DATA_BLOCK "FixReadCap_copy"
{ S7_Optimized_Access := 'FALSE' }
VERSION : 0.1
   STRUCT
      W0 : Int;   // M501_Z0 Destination_1A
      W2 : Int;   // M501_Z0 Destination_1B
      W4 : Int;   // M501_Z0 Destination_1C
      W6 : Int;   // M501_Z0 Destination_1D
      W8 : Int;   // M501_Z0 Length_1A (x) [dm]
      W10 : Int;   // M501_Z0 Length_1B (x) [dm]
      W12 : Int;   // M501_Z0 Length_1C (x) [dm]
      W14 : Int;   // M501_Z0 Length_1D (x) [dm]
      W16 : Int;   // M501_Z0 Width_1A  (y) [dm]
      W18 : Int;   // M501_Z0 Width_1B  (y) [dm]
      W20 : Int;   // M501_Z0 Width_1C  (y) [dm]
      W22 : Int;   // M501_Z0 Width_1D  (y) [dm]
      W24 : Int;   // M501_Z0 Position_X_1A  [dm]
      W26 : Int;   // M501_Z0 Position_X_1B  [dm]
      W28 : Int;   // M501_Z0 Position_X_1C  [dm]
      W30 : Int;   // M501_Z0 Position_X_1D  [dm]
      W32 : Int;   // M501_Z0 Position_Y_1A  [dm]
      W34 : Int;   // M501_Z0 Position_Y_1B  [dm]
      W36 : Int;   // M501_Z0 Position_Y_1C  [dm]
      W38 : Int;   // M501_Z0 Position_Y_1D  [dm]
      W40 : Int;   // M501_Z0 Code_1A_not used
      W42 : Int;   // M501_Z0 Code_1B_not used
      W44 : Int;   // M501_Z0 Code_1C_not used
      W46 : Int;   // M501_Z0 Code_1D_not used
      W48 : Int;
      W50 : Int;   // M501_Z1 Destination_1A
      W52 : Int;   // M501_Z1 Destination_1B
      W54 : Int;   // M501_Z1 Destination_1C
      W56 : Int;   // M501_Z1 Destination_1D
      W58 : Int;   // M501_Z1 Length_1A (x) [dm]
      W60 : Int;   // M501_Z1 Length_1B (x) [dm]
      W62 : Int;   // M501_Z1 Length_1C (x) [dm]
      W64 : Int;   // M501_Z1 Length_1D (x) [dm]
      W66 : Int;   // M501_Z1 Width_1A  (y) [dm]
      W68 : Int;   // M501_Z1 Width_1B  (y) [dm]
      W70 : Int;   // M501_Z1 Width_1C  (y) [dm]
      W72 : Int;   // M501_Z1 Width_1D  (y) [dm]
      W74 : Int;   // M501_Z1 Position_X_1A  [dm]
      W76 : Int;   // M501_Z1 Position_X_1B  [dm]
      W78 : Int;   // M501_Z1 Position_X_1C  [dm]
      W80 : Int;   // M501_Z1 Position_X_1D  [dm]
      W82 : Int;   // M501_Z1 Position_Y_1A  [dm]
      W84 : Int;   // M501_Z1 Position_Y_1B  [dm]
      W86 : Int;   // M501_Z1 Position_Y_1C  [dm]
      W88 : Int;   // M501_Z1 Position_Y_1D  [dm]
      W90 : Int;   // M501_Z1 Code_1A_not used
      W92 : Int;   // M501_Z1 Code_1B_not used
      W94 : Int;   // M501_Z1 Code_1C_not used
      W96 : Int;   // M501_Z1 Code_1D_not used
      W98 : Int;
      W100 : Int;   // M501_Z2 Destination_1A
      W102 : Int;   // M501_Z2 Destination_1B
      W104 : Int;   // M501_Z2 Destination_1C
      W106 : Int;   // M501_Z2 Destination_1D
      W108 : Int;   // M501_Z2 Length_1A (x) [dm]
      W110 : Int;   // M501_Z2 Length_1B (x) [dm]
      W112 : Int;   // M501_Z2 Length_1C (x) [dm]
      W114 : Int;   // M501_Z2 Length_1D (x) [dm]
      W116 : Int;   // M501_Z2 Width_1A  (y) [dm]
      W118 : Int;   // M501_Z2 Width_1B  (y) [dm]
      W120 : Int;   // M501_Z2 Width_1C  (y) [dm]
      W122 : Int;   // M501_Z2 Width_1D  (y) [dm]
      W124 : Int;   // M501_Z2 Position_X_1A  [dm]
      W126 : Int;   // M501_Z2 Position_X_1B  [dm]
      W128 : Int;   // M501_Z2 Position_X_1C  [dm]
      W130 : Int;   // M501_Z2 Position_X_1D  [dm]
      W132 : Int;   // M501_Z2 Position_Y_1A  [dm]
      W134 : Int;   // M501_Z2 Position_Y_1B  [dm]
      W136 : Int;   // M501_Z2 Position_Y_1C  [dm]
      W138 : Int;   // M501_Z2 Position_Y_1D  [dm]
      W140 : Int;   // M501_Z2 Code_1A_not used
      W142 : Int;   // M501_Z2 Code_1B_not used
      W144 : Int;   // M501_Z2 Code_1C_not used
      W146 : Int;   // M501_Z2 Code_1D_not used
      W148 : Int;
      W150 : Int;   // M319 Destination_1A
      W152 : Int;   // M319 Destination_2A
      W154 : Int;   // M319 Destination_3A
      W156 : Int;   // M319 Destination_4A
      W158 : Int;   // M319 Length_1A (x) [dm]
      W160 : Int;   // M319 Length_2A (x) [dm]
      W162 : Int;   // M319 Length_3A (x) [dm]
      W164 : Int;   // M319 Length_4A (x) [dm]
      W166 : Int;   // M319 Width_1A  (y) [dm]
      W168 : Int;   // M319 Width_2A  (y) [dm]
      W170 : Int;   // M319 Width_3A  (y) [dm]
      W172 : Int;   // M319 Width_4A  (y) [dm]
      W174 : Int;   // M319 Position_X_1A  [dm]
      W176 : Int;   // M319 Position_X_2A  [dm]
      W178 : Int;   // M319 Position_X_3A  [dm]
      W180 : Int;   // M319 Position_X_4A  [dm]
      W182 : Int;   // M319 Position_Y_1A  [dm]
      W184 : Int;   // M319 Position_Y_2A  [dm]
      W186 : Int;   // M319 Position_Y_3A  [dm]
      W188 : Int;   // M319 Position_Y_4A  [dm]
      W190 : Int;   // M319 Code_1A_not used
      W192 : Int;   // M319 Code_2A_not used
      W194 : Int;   // M319 Code_3A_not used
      W196 : Int;   // M319 Code_4A_not used
      W198 : Int;
      W200 : Int;   // M502 Destination_1A
      W202 : Int;   // M502 Destination_2A
      W204 : Int;   // M502 Destination_3A
      W206 : Int;   // M502 Destination_4A
      W208 : Int;   // M502 Length_1A (x) [dm]
      W210 : Int;   // M502 Length_2A (x) [dm]
      W212 : Int;   // M502 Length_3A (x) [dm]
      W214 : Int;   // M502 Length_4A (x) [dm]
      W216 : Int;   // M502 Width_1A  (y) [dm]
      W218 : Int;   // M502 Width_2A  (y) [dm]
      W220 : Int;   // M502 Width_3A  (y) [dm]
      W222 : Int;   // M502 Width_4A  (y) [dm]
      W224 : Int;   // M502 Position_X_1A  [dm]
      W226 : Int;   // M502 Position_X_2A  [dm]
      W228 : Int;   // M502 Position_X_3A  [dm]
      W230 : Int;   // M502 Position_X_4A  [dm]
      W232 : Int;   // M502 Position_Y_1A  [dm]
      W234 : Int;   // M502 Position_Y_2A  [dm]
      W236 : Int;   // M502 Position_Y_3A  [dm]
      W238 : Int;   // M502 Position_Y_4A  [dm]
      W240 : Int;   // M502 Code_1A_not used
      W242 : Int;   // M502 Code_2A_not used
      W244 : Int;   // M502 Code_3A_not used
      W246 : Int;   // M502 Code_4A_not used
      W248 : Int;
      W250 : Int;   // M502 Destination_1B
      W252 : Int;   // M502 Destination_2B
      W254 : Int;   // M502 Destination_3B
      W256 : Int;   // M502 Destination_4B
      W258 : Int;   // M502 Length_1B (x) [dm]
      W260 : Int;   // M502 Length_2B (x) [dm]
      W262 : Int;   // M502 Length_3B (x) [dm]
      W264 : Int;   // M502 Length_4B (x) [dm]
      W266 : Int;   // M502 Width_1B  (y) [dm]
      W268 : Int;   // M502 Width_2B  (y) [dm]
      W270 : Int;   // M502 Width_3B  (y) [dm]
      W272 : Int;   // M502 Width_4B  (y) [dm]
      W274 : Int;   // M502 Position_X_1B  [dm]
      W276 : Int;   // M502 Position_X_2B  [dm]
      W278 : Int;   // M502 Position_X_3B  [dm]
      W280 : Int;   // M502 Position_X_4B  [dm]
      W282 : Int;   // M502 Position_Y_1B  [dm]
      W284 : Int;   // M502 Position_Y_2B  [dm]
      W286 : Int;   // M502 Position_Y_3B  [dm]
      W288 : Int;   // M502 Position_Y_4B  [dm]
      W290 : Int;   // M502 Code_1B_not used
      W292 : Int;   // M502 Code_2B_not used
      W294 : Int;   // M502 Code_3B_not used
      W296 : Int;   // M502 Code_4B_not used
      W298 : Int;
      W300 : Int;   // M504 Destination_1A
      W302 : Int;   // M504 Destination_2A
      W304 : Int;   // M504 Destination_3A
      W306 : Int;   // M504 Destination_4A
      W308 : Int;   // M504 Length_1A (x) [dm]
      W310 : Int;   // M504 Length_2A (x) [dm]
      W312 : Int;   // M504 Length_3A (x) [dm]
      W314 : Int;   // M504 Length_4A (x) [dm]
      W316 : Int;   // M504 Width_1A  (y) [dm]
      W318 : Int;   // M504 Width_2A  (y) [dm]
      W320 : Int;   // M504 Width_3A  (y) [dm]
      W322 : Int;   // M504 Width_4A  (y) [dm]
      W324 : Int;   // M504 Position_X_1A  [dm]
      W326 : Int;   // M504 Position_X_2A  [dm]
      W328 : Int;   // M504 Position_X_3A  [dm]
      W330 : Int;   // M504 Position_X_4A  [dm]
      W332 : Int;   // M504 Position_Y_1A  [dm]
      W334 : Int;   // M504 Position_Y_2A  [dm]
      W336 : Int;   // M504 Position_Y_3A  [dm]
      W338 : Int;   // M504 Position_Y_4A  [dm]
      W340 : Int;   // M504 Code_1A_not used
      W342 : Int;   // M504 Code_2A_not used
      W344 : Int;   // M504 Code_3A_not used
      W346 : Int;   // M504 Code_4A_not used
      W348 : Int;
      W350 : Int;   // M504 Destination_1B
      W352 : Int;   // M504 Destination_2B
      W354 : Int;   // M504 Destination_3B
      W356 : Int;   // M504 Destination_4B
      W358 : Int;   // M504 Length_1B (x) [dm]
      W360 : Int;   // M504 Length_2B (x) [dm]
      W362 : Int;   // M504 Length_3B (x) [dm]
      W364 : Int;   // M504 Length_4B (x) [dm]
      W366 : Int;   // M504 Width_1B  (y) [dm]
      W368 : Int;   // M504 Width_2B  (y) [dm]
      W370 : Int;   // M504 Width_3B  (y) [dm]
      W372 : Int;   // M504 Width_4B  (y) [dm]
      W374 : Int;   // M504 Position_X_1B  [dm]
      W376 : Int;   // M504 Position_X_2B  [dm]
      W378 : Int;   // M504 Position_X_3B  [dm]
      W380 : Int;   // M504 Position_X_4B  [dm]
      W382 : Int;   // M504 Position_Y_1B  [dm]
      W384 : Int;   // M504 Position_Y_2B  [dm]
      W386 : Int;   // M504 Position_Y_3B  [dm]
      W388 : Int;   // M504 Position_Y_4B  [dm]
      W390 : Int;   // M504 Code_1B_not used
      W392 : Int;   // M504 Code_2B_not used
      W394 : Int;   // M504 Code_3B_not used
      W396 : Int;   // M504 Code_4B_not used
      W398 : Int;
      W400 : Int;   // M505 Destination_1A
      W402 : Int;   // M505 Destination_2A
      W404 : Int;   // M505 Destination_3A
      W406 : Int;   // M505 Destination_4A
      W408 : Int;   // M505 Length_1A (x) [dm]
      W410 : Int;   // M505 Length_2A (x) [dm]
      W412 : Int;   // M505 Length_3A (x) [dm]
      W414 : Int;   // M505 Length_4A (x) [dm]
      W416 : Int;   // M505 Width_1A  (y) [dm]
      W418 : Int;   // M505 Width_2A  (y) [dm]
      W420 : Int;   // M505 Width_3A  (y) [dm]
      W422 : Int;   // M505 Width_4A  (y) [dm]
      W424 : Int;   // M505 Position_X_1A  [dm]
      W426 : Int;   // M505 Position_X_2A  [dm]
      W428 : Int;   // M505 Position_X_3A  [dm]
      W430 : Int;   // M505 Position_X_4A  [dm]
      W432 : Int;   // M505 Position_Y_1A  [dm]
      W434 : Int;   // M505 Position_Y_2A  [dm]
      W436 : Int;   // M505 Position_Y_3A  [dm]
      W438 : Int;   // M505 Position_Y_4A  [dm]
      W440 : Int;   // M505 Code_1A_not used
      W442 : Int;   // M505 Code_2A_not used
      W444 : Int;   // M505 Code_3A_not used
      W446 : Int;   // M505 Code_4A_not used
      W448 : Int;
      W450 : Int;   // M505 Destination_1B
      W452 : Int;   // M505 Destination_2B
      W454 : Int;   // M505 Destination_3B
      W456 : Int;   // M505 Destination_4B
      W458 : Int;   // M505 Length_1B (x) [dm]
      W460 : Int;   // M505 Length_2B (x) [dm]
      W462 : Int;   // M505 Length_3B (x) [dm]
      W464 : Int;   // M505 Length_4B (x) [dm]
      W466 : Int;   // M505 Width_1B  (y) [dm]
      W468 : Int;   // M505 Width_2B  (y) [dm]
      W470 : Int;   // M505 Width_3B  (y) [dm]
      W472 : Int;   // M505 Width_4B  (y) [dm]
      W474 : Int;   // M505 Position_X_1B  [dm]
      W476 : Int;   // M505 Position_X_2B  [dm]
      W478 : Int;   // M505 Position_X_3B  [dm]
      W480 : Int;   // M505 Position_X_4B  [dm]
      W482 : Int;   // M505 Position_Y_1B  [dm]
      W484 : Int;   // M505 Position_Y_2B  [dm]
      W486 : Int;   // M505 Position_Y_3B  [dm]
      W488 : Int;   // M505 Position_Y_4B  [dm]
      W490 : Int;   // M505 Code_1B_not used
      W492 : Int;   // M505 Code_2B_not used
      W494 : Int;   // M505 Code_3B_not used
      W496 : Int;   // M505 Code_4B_not used
      W498 : Int;
      W500 : Int;   // M506 Destination_1A
      W502 : Int;   // M506 Destination_2A
      W504 : Int;   // M506 Destination_3A
      W506 : Int;   // M506 Destination_4A
      W508 : Int;   // M506 Length_1A (x) [dm]
      W510 : Int;   // M506 Length_2A (x) [dm]
      W512 : Int;   // M506 Length_3A (x) [dm]
      W514 : Int;   // M506 Length_4A (x) [dm]
      W516 : Int;   // M506 Width_1A  (y) [dm]
      W518 : Int;   // M506 Width_2A  (y) [dm]
      W520 : Int;   // M506 Width_3A  (y) [dm]
      W522 : Int;   // M506 Width_4A  (y) [dm]
      W524 : Int;   // M506 Position_X_1A  [dm]
      W526 : Int;   // M506 Position_X_2A  [dm]
      W528 : Int;   // M506 Position_X_3A  [dm]
      W530 : Int;   // M506 Position_X_4A  [dm]
      W532 : Int;   // M506 Position_Y_1A  [dm]
      W534 : Int;   // M506 Position_Y_2A  [dm]
      W536 : Int;   // M506 Position_Y_3A  [dm]
      W538 : Int;   // M506 Position_Y_4A  [dm]
      W540 : Int;   // M506 Code_1A_not used
      W542 : Int;   // M506 Code_2A_not used
      W544 : Int;   // M506 Code_3A_not used
      W546 : Int;   // M506 Code_4A_not used
      W548 : Int;
      W550 : Int;   // M506 Destination_1B
      W552 : Int;   // M506 Destination_2B
      W554 : Int;   // M506 Destination_3B
      W556 : Int;   // M506 Destination_4B
      W558 : Int;   // M506 Length_1B (x) [dm]
      W560 : Int;   // M506 Length_2B (x) [dm]
      W562 : Int;   // M506 Length_3B (x) [dm]
      W564 : Int;   // M506 Length_4B (x) [dm]
      W566 : Int;   // M506 Width_1B  (y) [dm]
      W568 : Int;   // M506 Width_2B  (y) [dm]
      W570 : Int;   // M506 Width_3B  (y) [dm]
      W572 : Int;   // M506 Width_4B  (y) [dm]
      W574 : Int;   // M506 Position_X_1B  [dm]
      W576 : Int;   // M506 Position_X_2B  [dm]
      W578 : Int;   // M506 Position_X_3B  [dm]
      W580 : Int;   // M506 Position_X_4B  [dm]
      W582 : Int;   // M506 Position_Y_1B  [dm]
      W584 : Int;   // M506 Position_Y_2B  [dm]
      W586 : Int;   // M506 Position_Y_3B  [dm]
      W588 : Int;   // M506 Position_Y_4B  [dm]
      W590 : Int;   // M506 Code_1B_not used
      W592 : Int;   // M506 Code_2B_not used
      W594 : Int;   // M506 Code_3B_not used
      W596 : Int;   // M506 Code_4B_not used
      W598 : Int;
      W600 : Int;
   END_STRUCT;


BEGIN
   W150 := 30;
   W158 := 36;
   W166 := 15;
   W168 := 15;
   W170 := 15;
   W172 := 15;
   W174 := 3;
   W176 := -34;
   W178 := -71;
   W180 := -108;
   W182 := 15;
   W184 := 15;
   W186 := 15;
   W188 := 15;
   W190 := 7255;
   W200 := 1;
   W206 := 30541;

END_DATA_BLOCK

DATA_BLOCK "FixReadCap"
{ S7_Optimized_Access := 'FALSE' }
VERSION : 0.1
   STRUCT
      W0 : Int;   // M501_Z0 Destination_1A
      W2 : Int;   // M501_Z0 Destination_1B
      W4 : Int;   // M501_Z0 Destination_1C
      W6 : Int;   // M501_Z0 Destination_1D
      W8 : Int;   // M501_Z0 Length_1A (x) [dm]
      W10 : Int;   // M501_Z0 Length_1B (x) [dm]
      W12 : Int;   // M501_Z0 Length_1C (x) [dm]
      W14 : Int;   // M501_Z0 Length_1D (x) [dm]
      W16 : Int;   // M501_Z0 Width_1A  (y) [dm]
      W18 : Int;   // M501_Z0 Width_1B  (y) [dm]
      W20 : Int;   // M501_Z0 Width_1C  (y) [dm]
      W22 : Int;   // M501_Z0 Width_1D  (y) [dm]
      W24 : Int;   // M501_Z0 Position_X_1A  [dm]
      W26 : Int;   // M501_Z0 Position_X_1B  [dm]
      W28 : Int;   // M501_Z0 Position_X_1C  [dm]
      W30 : Int;   // M501_Z0 Position_X_1D  [dm]
      W32 : Int;   // M501_Z0 Position_Y_1A  [dm]
      W34 : Int;   // M501_Z0 Position_Y_1B  [dm]
      W36 : Int;   // M501_Z0 Position_Y_1C  [dm]
      W38 : Int;   // M501_Z0 Position_Y_1D  [dm]
      W40 : Int;   // M501_Z0 Code_1A_not used
      W42 : Int;   // M501_Z0 Code_1B_not used
      W44 : Int;   // M501_Z0 Code_1C_not used
      W46 : Int;   // M501_Z0 Code_1D_not used
      W48 : Int;
      W50 : Int;   // M501_Z1 Destination_1A
      W52 : Int;   // M501_Z1 Destination_1B
      W54 : Int;   // M501_Z1 Destination_1C
      W56 : Int;   // M501_Z1 Destination_1D
      W58 : Int;   // M501_Z1 Length_1A (x) [dm]
      W60 : Int;   // M501_Z1 Length_1B (x) [dm]
      W62 : Int;   // M501_Z1 Length_1C (x) [dm]
      W64 : Int;   // M501_Z1 Length_1D (x) [dm]
      W66 : Int;   // M501_Z1 Width_1A  (y) [dm]
      W68 : Int;   // M501_Z1 Width_1B  (y) [dm]
      W70 : Int;   // M501_Z1 Width_1C  (y) [dm]
      W72 : Int;   // M501_Z1 Width_1D  (y) [dm]
      W74 : Int;   // M501_Z1 Position_X_1A  [dm]
      W76 : Int;   // M501_Z1 Position_X_1B  [dm]
      W78 : Int;   // M501_Z1 Position_X_1C  [dm]
      W80 : Int;   // M501_Z1 Position_X_1D  [dm]
      W82 : Int;   // M501_Z1 Position_Y_1A  [dm]
      W84 : Int;   // M501_Z1 Position_Y_1B  [dm]
      W86 : Int;   // M501_Z1 Position_Y_1C  [dm]
      W88 : Int;   // M501_Z1 Position_Y_1D  [dm]
      W90 : Int;   // M501_Z1 Code_1A_not used
      W92 : Int;   // M501_Z1 Code_1B_not used
      W94 : Int;   // M501_Z1 Code_1C_not used
      W96 : Int;   // M501_Z1 Code_1D_not used
      W98 : Int;
      W100 : Int;   // M501_Z2 Destination_1A
      W102 : Int;   // M501_Z2 Destination_1B
      W104 : Int;   // M501_Z2 Destination_1C
      W106 : Int;   // M501_Z2 Destination_1D
      W108 : Int;   // M501_Z2 Length_1A (x) [dm]
      W110 : Int;   // M501_Z2 Length_1B (x) [dm]
      W112 : Int;   // M501_Z2 Length_1C (x) [dm]
      W114 : Int;   // M501_Z2 Length_1D (x) [dm]
      W116 : Int;   // M501_Z2 Width_1A  (y) [dm]
      W118 : Int;   // M501_Z2 Width_1B  (y) [dm]
      W120 : Int;   // M501_Z2 Width_1C  (y) [dm]
      W122 : Int;   // M501_Z2 Width_1D  (y) [dm]
      W124 : Int;   // M501_Z2 Position_X_1A  [dm]
      W126 : Int;   // M501_Z2 Position_X_1B  [dm]
      W128 : Int;   // M501_Z2 Position_X_1C  [dm]
      W130 : Int;   // M501_Z2 Position_X_1D  [dm]
      W132 : Int;   // M501_Z2 Position_Y_1A  [dm]
      W134 : Int;   // M501_Z2 Position_Y_1B  [dm]
      W136 : Int;   // M501_Z2 Position_Y_1C  [dm]
      W138 : Int;   // M501_Z2 Position_Y_1D  [dm]
      W140 : Int;   // M501_Z2 Code_1A_not used
      W142 : Int;   // M501_Z2 Code_1B_not used
      W144 : Int;   // M501_Z2 Code_1C_not used
      W146 : Int;   // M501_Z2 Code_1D_not used
      W148 : Int;
      W150 : Int;   // M319 Destination_1A
      W152 : Int;   // M319 Destination_2A
      W154 : Int;   // M319 Destination_3A
      W156 : Int;   // M319 Destination_4A
      W158 : Int;   // M319 Length_1A (x) [dm]
      W160 : Int;   // M319 Length_2A (x) [dm]
      W162 : Int;   // M319 Length_3A (x) [dm]
      W164 : Int;   // M319 Length_4A (x) [dm]
      W166 : Int;   // M319 Width_1A  (y) [dm]
      W168 : Int;   // M319 Width_2A  (y) [dm]
      W170 : Int;   // M319 Width_3A  (y) [dm]
      W172 : Int;   // M319 Width_4A  (y) [dm]
      W174 : Int;   // M319 Position_X_1A  [dm]
      W176 : Int;   // M319 Position_X_2A  [dm]
      W178 : Int;   // M319 Position_X_3A  [dm]
      W180 : Int;   // M319 Position_X_4A  [dm]
      W182 : Int;   // M319 Position_Y_1A  [dm]
      W184 : Int;   // M319 Position_Y_2A  [dm]
      W186 : Int;   // M319 Position_Y_3A  [dm]
      W188 : Int;   // M319 Position_Y_4A  [dm]
      W190 : Int;   // M319 Code_1A_not used
      W192 : Int;   // M319 Code_2A_not used
      W194 : Int;   // M319 Code_3A_not used
      W196 : Int;   // M319 Code_4A_not used
      W198 : Int;
      W200 : Int;   // M502 Destination_1A
      W202 : Int;   // M502 Destination_2A
      W204 : Int;   // M502 Destination_3A
      W206 : Int;   // M502 Destination_4A
      W208 : Int;   // M502 Length_1A (x) [dm]
      W210 : Int;   // M502 Length_2A (x) [dm]
      W212 : Int;   // M502 Length_3A (x) [dm]
      W214 : Int;   // M502 Length_4A (x) [dm]
      W216 : Int;   // M502 Width_1A  (y) [dm]
      W218 : Int;   // M502 Width_2A  (y) [dm]
      W220 : Int;   // M502 Width_3A  (y) [dm]
      W222 : Int;   // M502 Width_4A  (y) [dm]
      W224 : Int;   // M502 Position_X_1A  [dm]
      W226 : Int;   // M502 Position_X_2A  [dm]
      W228 : Int;   // M502 Position_X_3A  [dm]
      W230 : Int;   // M502 Position_X_4A  [dm]
      W232 : Int;   // M502 Position_Y_1A  [dm]
      W234 : Int;   // M502 Position_Y_2A  [dm]
      W236 : Int;   // M502 Position_Y_3A  [dm]
      W238 : Int;   // M502 Position_Y_4A  [dm]
      W240 : Int;   // M502 Code_1A_not used
      W242 : Int;   // M502 Code_2A_not used
      W244 : Int;   // M502 Code_3A_not used
      W246 : Int;   // M502 Code_4A_not used
      W248 : Int;
      W250 : Int;   // M502 Destination_1B
      W252 : Int;   // M502 Destination_2B
      W254 : Int;   // M502 Destination_3B
      W256 : Int;   // M502 Destination_4B
      W258 : Int;   // M502 Length_1B (x) [dm]
      W260 : Int;   // M502 Length_2B (x) [dm]
      W262 : Int;   // M502 Length_3B (x) [dm]
      W264 : Int;   // M502 Length_4B (x) [dm]
      W266 : Int;   // M502 Width_1B  (y) [dm]
      W268 : Int;   // M502 Width_2B  (y) [dm]
      W270 : Int;   // M502 Width_3B  (y) [dm]
      W272 : Int;   // M502 Width_4B  (y) [dm]
      W274 : Int;   // M502 Position_X_1B  [dm]
      W276 : Int;   // M502 Position_X_2B  [dm]
      W278 : Int;   // M502 Position_X_3B  [dm]
      W280 : Int;   // M502 Position_X_4B  [dm]
      W282 : Int;   // M502 Position_Y_1B  [dm]
      W284 : Int;   // M502 Position_Y_2B  [dm]
      W286 : Int;   // M502 Position_Y_3B  [dm]
      W288 : Int;   // M502 Position_Y_4B  [dm]
      W290 : Int;   // M502 Code_1B_not used
      W292 : Int;   // M502 Code_2B_not used
      W294 : Int;   // M502 Code_3B_not used
      W296 : Int;   // M502 Code_4B_not used
      W298 : Int;
      W300 : Int;   // M504 Destination_1A
      W302 : Int;   // M504 Destination_2A
      W304 : Int;   // M504 Destination_3A
      W306 : Int;   // M504 Destination_4A
      W308 : Int;   // M504 Length_1A (x) [dm]
      W310 : Int;   // M504 Length_2A (x) [dm]
      W312 : Int;   // M504 Length_3A (x) [dm]
      W314 : Int;   // M504 Length_4A (x) [dm]
      W316 : Int;   // M504 Width_1A  (y) [dm]
      W318 : Int;   // M504 Width_2A  (y) [dm]
      W320 : Int;   // M504 Width_3A  (y) [dm]
      W322 : Int;   // M504 Width_4A  (y) [dm]
      W324 : Int;   // M504 Position_X_1A  [dm]
      W326 : Int;   // M504 Position_X_2A  [dm]
      W328 : Int;   // M504 Position_X_3A  [dm]
      W330 : Int;   // M504 Position_X_4A  [dm]
      W332 : Int;   // M504 Position_Y_1A  [dm]
      W334 : Int;   // M504 Position_Y_2A  [dm]
      W336 : Int;   // M504 Position_Y_3A  [dm]
      W338 : Int;   // M504 Position_Y_4A  [dm]
      W340 : Int;   // M504 Code_1A_not used
      W342 : Int;   // M504 Code_2A_not used
      W344 : Int;   // M504 Code_3A_not used
      W346 : Int;   // M504 Code_4A_not used
      W348 : Int;
      W350 : Int;   // M504 Destination_1B
      W352 : Int;   // M504 Destination_2B
      W354 : Int;   // M504 Destination_3B
      W356 : Int;   // M504 Destination_4B
      W358 : Int;   // M504 Length_1B (x) [dm]
      W360 : Int;   // M504 Length_2B (x) [dm]
      W362 : Int;   // M504 Length_3B (x) [dm]
      W364 : Int;   // M504 Length_4B (x) [dm]
      W366 : Int;   // M504 Width_1B  (y) [dm]
      W368 : Int;   // M504 Width_2B  (y) [dm]
      W370 : Int;   // M504 Width_3B  (y) [dm]
      W372 : Int;   // M504 Width_4B  (y) [dm]
      W374 : Int;   // M504 Position_X_1B  [dm]
      W376 : Int;   // M504 Position_X_2B  [dm]
      W378 : Int;   // M504 Position_X_3B  [dm]
      W380 : Int;   // M504 Position_X_4B  [dm]
      W382 : Int;   // M504 Position_Y_1B  [dm]
      W384 : Int;   // M504 Position_Y_2B  [dm]
      W386 : Int;   // M504 Position_Y_3B  [dm]
      W388 : Int;   // M504 Position_Y_4B  [dm]
      W390 : Int;   // M504 Code_1B_not used
      W392 : Int;   // M504 Code_2B_not used
      W394 : Int;   // M504 Code_3B_not used
      W396 : Int;   // M504 Code_4B_not used
      W398 : Int;
      W400 : Int;   // M505 Destination_1A
      W402 : Int;   // M505 Destination_2A
      W404 : Int;   // M505 Destination_3A
      W406 : Int;   // M505 Destination_4A
      W408 : Int;   // M505 Length_1A (x) [dm]
      W410 : Int;   // M505 Length_2A (x) [dm]
      W412 : Int;   // M505 Length_3A (x) [dm]
      W414 : Int;   // M505 Length_4A (x) [dm]
      W416 : Int;   // M505 Width_1A  (y) [dm]
      W418 : Int;   // M505 Width_2A  (y) [dm]
      W420 : Int;   // M505 Width_3A  (y) [dm]
      W422 : Int;   // M505 Width_4A  (y) [dm]
      W424 : Int;   // M505 Position_X_1A  [dm]
      W426 : Int;   // M505 Position_X_2A  [dm]
      W428 : Int;   // M505 Position_X_3A  [dm]
      W430 : Int;   // M505 Position_X_4A  [dm]
      W432 : Int;   // M505 Position_Y_1A  [dm]
      W434 : Int;   // M505 Position_Y_2A  [dm]
      W436 : Int;   // M505 Position_Y_3A  [dm]
      W438 : Int;   // M505 Position_Y_4A  [dm]
      W440 : Int;   // M505 Code_1A_not used
      W442 : Int;   // M505 Code_2A_not used
      W444 : Int;   // M505 Code_3A_not used
      W446 : Int;   // M505 Code_4A_not used
      W448 : Int;
      W450 : Int;   // M505 Destination_1B
      W452 : Int;   // M505 Destination_2B
      W454 : Int;   // M505 Destination_3B
      W456 : Int;   // M505 Destination_4B
      W458 : Int;   // M505 Length_1B (x) [dm]
      W460 : Int;   // M505 Length_2B (x) [dm]
      W462 : Int;   // M505 Length_3B (x) [dm]
      W464 : Int;   // M505 Length_4B (x) [dm]
      W466 : Int;   // M505 Width_1B  (y) [dm]
      W468 : Int;   // M505 Width_2B  (y) [dm]
      W470 : Int;   // M505 Width_3B  (y) [dm]
      W472 : Int;   // M505 Width_4B  (y) [dm]
      W474 : Int;   // M505 Position_X_1B  [dm]
      W476 : Int;   // M505 Position_X_2B  [dm]
      W478 : Int;   // M505 Position_X_3B  [dm]
      W480 : Int;   // M505 Position_X_4B  [dm]
      W482 : Int;   // M505 Position_Y_1B  [dm]
      W484 : Int;   // M505 Position_Y_2B  [dm]
      W486 : Int;   // M505 Position_Y_3B  [dm]
      W488 : Int;   // M505 Position_Y_4B  [dm]
      W490 : Int;   // M505 Code_1B_not used
      W492 : Int;   // M505 Code_2B_not used
      W494 : Int;   // M505 Code_3B_not used
      W496 : Int;   // M505 Code_4B_not used
      W498 : Int;
      W500 : Int;   // M506 Destination_1A
      W502 : Int;   // M506 Destination_2A
      W504 : Int;   // M506 Destination_3A
      W506 : Int;   // M506 Destination_4A
      W508 : Int;   // M506 Length_1A (x) [dm]
      W510 : Int;   // M506 Length_2A (x) [dm]
      W512 : Int;   // M506 Length_3A (x) [dm]
      W514 : Int;   // M506 Length_4A (x) [dm]
      W516 : Int;   // M506 Width_1A  (y) [dm]
      W518 : Int;   // M506 Width_2A  (y) [dm]
      W520 : Int;   // M506 Width_3A  (y) [dm]
      W522 : Int;   // M506 Width_4A  (y) [dm]
      W524 : Int;   // M506 Position_X_1A  [dm]
      W526 : Int;   // M506 Position_X_2A  [dm]
      W528 : Int;   // M506 Position_X_3A  [dm]
      W530 : Int;   // M506 Position_X_4A  [dm]
      W532 : Int;   // M506 Position_Y_1A  [dm]
      W534 : Int;   // M506 Position_Y_2A  [dm]
      W536 : Int;   // M506 Position_Y_3A  [dm]
      W538 : Int;   // M506 Position_Y_4A  [dm]
      W540 : Int;   // M506 Code_1A_not used
      W542 : Int;   // M506 Code_2A_not used
      W544 : Int;   // M506 Code_3A_not used
      W546 : Int;   // M506 Code_4A_not used
      W548 : Int;
      W550 : Int;   // M506 Destination_1B
      W552 : Int;   // M506 Destination_2B
      W554 : Int;   // M506 Destination_3B
      W556 : Int;   // M506 Destination_4B
      W558 : Int;   // M506 Length_1B (x) [dm]
      W560 : Int;   // M506 Length_2B (x) [dm]
      W562 : Int;   // M506 Length_3B (x) [dm]
      W564 : Int;   // M506 Length_4B (x) [dm]
      W566 : Int;   // M506 Width_1B  (y) [dm]
      W568 : Int;   // M506 Width_2B  (y) [dm]
      W570 : Int;   // M506 Width_3B  (y) [dm]
      W572 : Int;   // M506 Width_4B  (y) [dm]
      W574 : Int;   // M506 Position_X_1B  [dm]
      W576 : Int;   // M506 Position_X_2B  [dm]
      W578 : Int;   // M506 Position_X_3B  [dm]
      W580 : Int;   // M506 Position_X_4B  [dm]
      W582 : Int;   // M506 Position_Y_1B  [dm]
      W584 : Int;   // M506 Position_Y_2B  [dm]
      W586 : Int;   // M506 Position_Y_3B  [dm]
      W588 : Int;   // M506 Position_Y_4B  [dm]
      W590 : Int;   // M506 Code_1B_not used
      W592 : Int;   // M506 Code_2B_not used
      W594 : Int;   // M506 Code_3B_not used
      W596 : Int;   // M506 Code_4B_not used
      W598 : Int;
      W600 : Int;
   END_STRUCT;


BEGIN
   W150 := 30;
   W158 := 36;
   W166 := 15;
   W168 := 15;
   W170 := 15;
   W172 := 15;
   W174 := 3;
   W176 := -34;
   W178 := -71;
   W180 := -108;
   W182 := 15;
   W184 := 15;
   W186 := 15;
   W188 := 15;
   W190 := 7255;
   W200 := 1;
   W206 := 30541;

END_DATA_BLOCK

DATA_BLOCK "DB_FixManComConv"
{ S7_Optimized_Access := 'FALSE' }
VERSION : 0.0
   STRUCT
      b00 : Bool;
      b01 : Bool;
      b02 : Bool;
      b03 : Bool;
      b04 : Bool;
      b05 : Bool;
      b06 : Bool;
      b07 : Bool;
      b10 : Bool;
      b11 : Bool;
      b12 : Bool;
      b13 : Bool;
      b14 : Bool;
      b15 : Bool;
      b16 : Bool;
      b17 : Bool;
      b20 : Bool;
      b21 : Bool;
      b22 : Bool;
      b23 : Bool;
      b24 : Bool;
      b25 : Bool;
      b26 : Bool;
      b27 : Bool;
      b30 : Bool;
      b31 : Bool;
      b32 : Bool;
      b33 : Bool;
      b34 : Bool;
      b35 : Bool;
      b36 : Bool;
      b37 : Bool;
      b40 : Bool;   // M501_M1 p.b.:rollers rotation forward (M.L.D.)
      b41 : Bool;   // M501_M1 p.b.:rollers rotation backward (M.L.D.)
      b42 : Bool;   // M501_M2 p.b.:wheels zone 1 rotation forward (M.L.D.)
      b43 : Bool;   // M501_M2 p.b.:wheels zone 1 rotation backward (M.L.D.)
      b44 : Bool;   // M501_M3 p.b.:wheels zone 2 rotation forward (M.L.D.)
      b45 : Bool;   // M501_M3 p.b.:wheels zone 2 rotation backward (M.L.D.)
      b46 : Bool;   // M501_M2-3 p.b.:wheels zone 1-2 rotation forward (M.L.D.)
      b47 : Bool;   // M501_M2-3 p.b.:wheels zone 1-2 rotation backward (M.L.D.)
      b50 : Bool;   // M501_M1-2-3 p.b.:rollers and wheels zone 1-2 rotation forward (M.L.D.)
      b51 : Bool;   // M501_M1-2-3 p.b.:rollers and wheels zone 1-2 rotation backward (M.L.D.)
      PF_M501 : Bool;   // M501_M4 p.b.:small wheels rotation forward (L.L.D.)
      PB_M501 : Bool;   // M501_M4 p.b.:small wheels rotation backward (L.L.D.)
      b54 : Bool;
      b55 : Bool;
      b56 : Bool;   // M501_M4M5 p.b.:raise small wheels chassis
      b57 : Bool;   // M501_M4M5 p.b.:descent small wheels chassis
      PF_M502 : Bool;   // M502_M1 p.b.:rollers rotation forward
      PB_M502 : Bool;   // M502_M1 p.b.:rollers rotation backward
      b62 : Bool;
      b63 : Bool;
      b64 : Bool;
      b65 : Bool;
      b66 : Bool;
      b67 : Bool;
      b70 : Bool;
      b71 : Bool;
      b72 : Bool;
      b73 : Bool;
      b74 : Bool;
      b75 : Bool;
      b76 : Bool;
      b77 : Bool;
      b80 : Bool;   // M503_M1 p.b.:Forward rotation (CW) Rotator Frame
      b81 : Bool;   // M503_M1 p.b.:Backward rotation (CCW) Rotator Frame
      b82 : Bool;   // //M503. p.b.: Raise of Rotator frame
      b83 : Bool;   // //M503. p.b.: Descent of Rotator frame
      b84 : Bool;   // //M503. p.b.: Centering device insertion
      b85 : Bool;   // //M503. p.b.: Centering device extraction
      b86 : Bool;
      b87 : Bool;
      b90 : Bool;
      b91 : Bool;
      b92 : Bool;
      b93 : Bool;
      b94 : Bool;
      b95 : Bool;
      b96 : Bool;
      b97 : Bool;
      PF_M504B : Bool;   // M504_M1 p.b.:rollers rotation forward
      PB_M504B : Bool;   // M504_M1 p.b.:rollers rotation backward
      PF_M504A : Bool;   // M504_M2 p.b.:rollers rotation forward
      PB_M504A : Bool;   // M504_M2 p.b.:rollers rotation backward
      PF_M504AB : Bool;   // M504_M1-2 p.b.:wheels zone 1-2 rotation forward
      PB_M504AB : Bool;   // M504_M1-2 p.b.:wheels zone 1-2 rotation backward
      b106 : Bool;
      b107 : Bool;
      b110 : Bool;
      b111 : Bool;
      b112 : Bool;
      b113 : Bool;
      b114 : Bool;
      b115 : Bool;
      b116 : Bool;
      b117 : Bool;
      PF_M505B : Bool;   // M505_M1 p.b.:rollers rotation forward
      PB_M505B : Bool;   // M505_M1 p.b.:rollers rotation backward
      PF_M505A : Bool;   // M505_M2 p.b.:rollers rotation forward
      PB_M505A : Bool;   // M505_M2 p.b.:rollers rotation backward
      PF_M505AB : Bool;   // M505_M1-2 p.b.:wheels zone 1-2 rotation forward
      PB_M505AB : Bool;   // M505_M1-2 p.b.:wheels zone 1-2 rotation backward
      PF_M505BSQ : Bool;   // M505_M1 p.b.:squaring raise and rollers rotation forward at squaring speed
      PF_M505ASQ : Bool;   // M505_M2 p.b.:squaring raise and rollers rotation forward at squaring speed
      PF_M505SQ : Bool;   // M505_M1-2 p.b.:squaring raise and rollers rot. 1-2 forward at squar. speed
      b131 : Bool;
      b132 : Bool;
      b133 : Bool;
      b134 : Bool;
      b135 : Bool;
      b136 : Bool;
      b137 : Bool;
      PF_M506B : Bool;   // M506_M1 p.b.:rollers rotation forward (LLD)
      PB_M506B : Bool;   // M506_M1 p.b.:rollers rotation backward (LLD)
      PF_M506A : Bool;   // M506_M2 p.b.:rollers rotation forward (LLD)
      PB_M506A : Bool;   // M506_M2 p.b.:rollers rotation backward (LLD)
      PF_M506AB : Bool;   // M506_M1-2 p.b.:wheels zone 1-2 rotation forward (LLD)
      PB_M506AB : Bool;   // M506_M1-2 p.b.:wheels zone 1-2 rotation backward (LLD)
      b146 : Bool;   // M506 p.b.:raise wheels chassis
      b147 : Bool;   // M506 p.b.:descent wheels chassis
      PL_M506B : Bool;   // M506_M3 p.b.:rollers rotation left (MLD)
      PR_M506B : Bool;   // M506_M3 p.b.:rollers rotation right (MLD)
      PL_M506A : Bool;   // M506_M4 p.b.:rollers rotation left (MLD)
      PR_M506A : Bool;   // M506_M4 p.b.:rollers rotation right (MLD)
      PL_M506AB : Bool;   // M506_M3-4 p.b.:rollers rotation left (MLD)
      PR_M506AB : Bool;   // M506_M3-4 p.b.:rollers rotation right (MLD)
      b156 : Bool;
      b157 : Bool;
      PF_M501_M502 : Bool;   // M501_M502 p.b.:rollers rotation forward (LLD)
      PB_M501_M502 : Bool;   // M501_M502 p.b.:rollers rotation backward (LLD)
      PF_M502_M504 : Bool;   // M502_M504 p.b.:rollers rotation forward
      PB_M502_M504 : Bool;   // M502_M504 p.b.:rollers rotation backward
      PF_M504_M505 : Bool;   // M504_M505 p.b.:rollers rotation forward
      PB_M504_M505 : Bool;   // M504_M505 p.b.:rollers rotation backward
      PF_M505_M506 : Bool;   // M505_M506 p.b.:rollers rotation Forward
      PB_M505_M506 : Bool;   // M505_M506 p.b.:rollers rotation backward
      b170 : Bool;   // M501 p.b all motors forward (MLD)
      b171 : Bool;   // M501 p.b all motors backward (MLD)
      PF_ALL : Bool;   // M501_M506 p.b all motors forward (LLD)
      PB_ALL : Bool;   // M501_M506 p.b all motors backward (LLD)
      b174 : Bool;
      b175 : Bool;
      b176 : Bool;
      b177 : Bool;
      P_M506_M6_L : Bool;   // M506_M6 p.b.:move Left Photocell to the left
      P_M506_M6_R : Bool;   // M506_M6 p.b.:move Left Photocell to the right
      P_M506_M7_L : Bool;   // M506_M7 p.b.:move Right Photocell to the left
      P_M506_M7_R : Bool;   // M506_M7 p.b.:move Right Photocell to the right
      b184 : Bool;
      b185 : Bool;
      b186 : Bool;
      b187 : Bool;
      b190 : Bool;
      b191 : Bool;
      b192 : Bool;
      b193 : Bool;
      b194 : Bool;
      b195 : Bool;
      b196 : Bool;
      b197 : Bool;
      b200 : Bool;
      b201 : Bool;
      b202 : Bool;
      b203 : Bool;
      b204 : Bool;
      b205 : Bool;
      b206 : Bool;
      b207 : Bool;
      b210 : Bool;
      b211 : Bool;
      b212 : Bool;
      b213 : Bool;
      b214 : Bool;
      b215 : Bool;
      b216 : Bool;
      b217 : Bool;
      b220 : Bool;
      b221 : Bool;
      b222 : Bool;
      b223 : Bool;
      b224 : Bool;
      b225 : Bool;
      b226 : Bool;
      b227 : Bool;
      b230 : Bool;
      b231 : Bool;
      b232 : Bool;
      b233 : Bool;
      b234 : Bool;
      b235 : Bool;
      b236 : Bool;
      b237 : Bool;
      b240 : Bool;
      b241 : Bool;
      b242 : Bool;
      b243 : Bool;
      b244 : Bool;
      b245 : Bool;
      b246 : Bool;
      b247 : Bool;
      b250 : Bool;
      b251 : Bool;
      b252 : Bool;
      b253 : Bool;
      b254 : Bool;
      b255 : Bool;
      b256 : Bool;
      b257 : Bool;
      b260 : Bool;
      b261 : Bool;
      b262 : Bool;
      b263 : Bool;
      b264 : Bool;
      b265 : Bool;
      b266 : Bool;
      b267 : Bool;
      b270 : Bool;
      b271 : Bool;
      b272 : Bool;
      b273 : Bool;
      b274 : Bool;
      b275 : Bool;
      b276 : Bool;
      b277 : Bool;
      b280 : Bool;
      b281 : Bool;
      b282 : Bool;
      b283 : Bool;
      b284 : Bool;
      b285 : Bool;
      b286 : Bool;
      b287 : Bool;
      b290 : Bool;
      b291 : Bool;
      b292 : Bool;
      b293 : Bool;
      b294 : Bool;
      b295 : Bool;
      b296 : Bool;
      b297 : Bool;
      b300 : Bool;
      b301 : Bool;
      b302 : Bool;
      b303 : Bool;
      b304 : Bool;
      b305 : Bool;
      b306 : Bool;
      b307 : Bool;
      b310 : Bool;
      b311 : Bool;
      b312 : Bool;
      b313 : Bool;
      b314 : Bool;
      b315 : Bool;
      b316 : Bool;
      b317 : Bool;
      b320 : Bool;
      b321 : Bool;
      b322 : Bool;
      b323 : Bool;
      b324 : Bool;
      b325 : Bool;
      b326 : Bool;
      b327 : Bool;
      b330 : Bool;
      b331 : Bool;
      b332 : Bool;
      b333 : Bool;
      b334 : Bool;
      b335 : Bool;
      b336 : Bool;
      b337 : Bool;
      b340 : Bool;
      b341 : Bool;
      b342 : Bool;
      b343 : Bool;
      b344 : Bool;
      b345 : Bool;
      b346 : Bool;
      b347 : Bool;
      b350 : Bool;
      b351 : Bool;
      b352 : Bool;
      b353 : Bool;
      b354 : Bool;
      b355 : Bool;
      b356 : Bool;
      b357 : Bool;
      b360 : Bool;
      b361 : Bool;
      b362 : Bool;
      b363 : Bool;
      b364 : Bool;
      b365 : Bool;
      b366 : Bool;
      b367 : Bool;
      b370 : Bool;
      b371 : Bool;
      b372 : Bool;
      b373 : Bool;
      b374 : Bool;
      b375 : Bool;
      b376 : Bool;
      b377 : Bool;
      b380 : Bool;
      b381 : Bool;
      b382 : Bool;
      b383 : Bool;
      b384 : Bool;
      b385 : Bool;
      b386 : Bool;
      b387 : Bool;
      b390 : Bool;
      b391 : Bool;
      b392 : Bool;
      b393 : Bool;
      b394 : Bool;
      b395 : Bool;
      b396 : Bool;
      b397 : Bool;
      b400 : Bool;
      b401 : Bool;
      b402 : Bool;
      b403 : Bool;
      b404 : Bool;
      b405 : Bool;
      b406 : Bool;
      b407 : Bool;
      b410 : Bool;
      b411 : Bool;
      b412 : Bool;
      b413 : Bool;
      b414 : Bool;
      b415 : Bool;
      b416 : Bool;
      b417 : Bool;
      b420 : Bool;
      b421 : Bool;
      b422 : Bool;
      b423 : Bool;
      b424 : Bool;
      b425 : Bool;
      b426 : Bool;
      b427 : Bool;
      b430 : Bool;
      b431 : Bool;
      b432 : Bool;
      b433 : Bool;
      b434 : Bool;
      b435 : Bool;
      b436 : Bool;
      b437 : Bool;
      b440 : Bool;
      b441 : Bool;
      b442 : Bool;
      b443 : Bool;
      b444 : Bool;
      b445 : Bool;
      b446 : Bool;
      b447 : Bool;
      b450 : Bool;
      b451 : Bool;
      b452 : Bool;
      b453 : Bool;
      b454 : Bool;
      b455 : Bool;
      b456 : Bool;
      b457 : Bool;
      b460 : Bool;
      b461 : Bool;
      b462 : Bool;
      b463 : Bool;
      b464 : Bool;
      b465 : Bool;
      b466 : Bool;
      b467 : Bool;
      b470 : Bool;
      b471 : Bool;
      b472 : Bool;
      b473 : Bool;
      b474 : Bool;
      b475 : Bool;
      b476 : Bool;
      b477 : Bool;
      b480 : Bool;
      b481 : Bool;
      b482 : Bool;
      b483 : Bool;
      b484 : Bool;
      b485 : Bool;
      b486 : Bool;
      b487 : Bool;
      b490 : Bool;
      b491 : Bool;
      b492 : Bool;
      b493 : Bool;
      b494 : Bool;
      b495 : Bool;
      b496 : Bool;
      b497 : Bool;
      b500 : Bool;
      b501 : Bool;
      b502 : Bool;
      b503 : Bool;
      b504 : Bool;
      b505 : Bool;
      b506 : Bool;
      b507 : Bool;
      b510 : Bool;
      b511 : Bool;
      b512 : Bool;
      b513 : Bool;
      b514 : Bool;
      b515 : Bool;
      b516 : Bool;
      b517 : Bool;
      b520 : Bool;
      b521 : Bool;
      b522 : Bool;
      b523 : Bool;
      b524 : Bool;
      b525 : Bool;
      b526 : Bool;
      b527 : Bool;
      b530 : Bool;
      b531 : Bool;
      b532 : Bool;
      b533 : Bool;
      b534 : Bool;
      b535 : Bool;
      b536 : Bool;
      b537 : Bool;
      b540 : Bool;
      b541 : Bool;
      b542 : Bool;
      b543 : Bool;
      b544 : Bool;
      b545 : Bool;
      b546 : Bool;
      b547 : Bool;
      b550 : Bool;
      b551 : Bool;
      b552 : Bool;
      b553 : Bool;
      b554 : Bool;
      b555 : Bool;
      b556 : Bool;
      b557 : Bool;
      b560 : Bool;
      b561 : Bool;
      b562 : Bool;
      b563 : Bool;
      b564 : Bool;
      b565 : Bool;
      b566 : Bool;
      b567 : Bool;
      b570 : Bool;
      b571 : Bool;
      b572 : Bool;
      b573 : Bool;
      b574 : Bool;
      b575 : Bool;
      b576 : Bool;
      b577 : Bool;
      b580 : Bool;
      b581 : Bool;
      b582 : Bool;
      b583 : Bool;
      b584 : Bool;
      b585 : Bool;
      b586 : Bool;
      b587 : Bool;
      b590 : Bool;
      b591 : Bool;
      b592 : Bool;
      b593 : Bool;
      b594 : Bool;
      b595 : Bool;
      b596 : Bool;
      b597 : Bool;
      b600 : Bool;
      b601 : Bool;
      b602 : Bool;
      b603 : Bool;
      b604 : Bool;
      b605 : Bool;
      b606 : Bool;
      b607 : Bool;
      b610 : Bool;
      b611 : Bool;
      b612 : Bool;
      b613 : Bool;
      b614 : Bool;
      b615 : Bool;
      b616 : Bool;
      b617 : Bool;
      b620 : Bool;
      b621 : Bool;
      b622 : Bool;
      b623 : Bool;
      b624 : Bool;
      b625 : Bool;
      b626 : Bool;
      b627 : Bool;
      b630 : Bool;
      b631 : Bool;
      b632 : Bool;
      b633 : Bool;
      b634 : Bool;
      b635 : Bool;
      b636 : Bool;
      b637 : Bool;
      b640 : Bool;
      b641 : Bool;
      b642 : Bool;
      b643 : Bool;
      b644 : Bool;
      b645 : Bool;
      b646 : Bool;
      b647 : Bool;
      b650 : Bool;
      b651 : Bool;
      b652 : Bool;
      b653 : Bool;
      b654 : Bool;
      b655 : Bool;
      b656 : Bool;
      b657 : Bool;
      b660 : Bool;
      b661 : Bool;
      b662 : Bool;
      b663 : Bool;
      b664 : Bool;
      b665 : Bool;
      b666 : Bool;
      b667 : Bool;
      b670 : Bool;
      b671 : Bool;
      b672 : Bool;
      b673 : Bool;
      b674 : Bool;
      b675 : Bool;
      b676 : Bool;
      b677 : Bool;
      b680 : Bool;
      b681 : Bool;
      b682 : Bool;
      b683 : Bool;
      b684 : Bool;
      b685 : Bool;
      b686 : Bool;
      b687 : Bool;
      b690 : Bool;
      b691 : Bool;
      b692 : Bool;
      b693 : Bool;
      b694 : Bool;
      b695 : Bool;
      b696 : Bool;
      b697 : Bool;
      b700 : Bool;
      b701 : Bool;
      b702 : Bool;
      b703 : Bool;
      b704 : Bool;
      b705 : Bool;
      b706 : Bool;
      b707 : Bool;
      b710 : Bool;
      b711 : Bool;
      b712 : Bool;
      b713 : Bool;
      b714 : Bool;
      b715 : Bool;
      b716 : Bool;
      b717 : Bool;
      b720 : Bool;
      b721 : Bool;
      b722 : Bool;
      b723 : Bool;
      b724 : Bool;
      b725 : Bool;
      b726 : Bool;
      b727 : Bool;
      b730 : Bool;
      b731 : Bool;
      b732 : Bool;
      b733 : Bool;
      b734 : Bool;
      b735 : Bool;
      b736 : Bool;
      b737 : Bool;
      b740 : Bool;
      b741 : Bool;
      b742 : Bool;
      b743 : Bool;
      b744 : Bool;
      b745 : Bool;
      b746 : Bool;
      b747 : Bool;
      b750 : Bool;
      b751 : Bool;
      b752 : Bool;
      b753 : Bool;
      b754 : Bool;
      b755 : Bool;
      b756 : Bool;
      b757 : Bool;
      b760 : Bool;
      b761 : Bool;
      b762 : Bool;
      b763 : Bool;
      b764 : Bool;
      b765 : Bool;
      b766 : Bool;
      b767 : Bool;
      b770 : Bool;
      b771 : Bool;
      b772 : Bool;
      b773 : Bool;
      b774 : Bool;
      b775 : Bool;
      b776 : Bool;
      b777 : Bool;
      b780 : Bool;
      b781 : Bool;
      b782 : Bool;
      b783 : Bool;
      b784 : Bool;
      b785 : Bool;
      b786 : Bool;
      b787 : Bool;
      b79 : Bool;
      b791 : Bool;
      b792 : Bool;
      b793 : Bool;
      b794 : Bool;
      b795 : Bool;
      b796 : Bool;
      b797 : Bool;
      b800 : Bool;
      b801 : Bool;
      b802 : Bool;
      b803 : Bool;
      b804 : Bool;
      b805 : Bool;
      b806 : Bool;
      b807 : Bool;
      b810 : Bool;
      b811 : Bool;
      b812 : Bool;
      b813 : Bool;
      b814 : Bool;
      b815 : Bool;
      b816 : Bool;
      b817 : Bool;
      b820 : Bool;
      b821 : Bool;
      b822 : Bool;
      b823 : Bool;
      b824 : Bool;
      b825 : Bool;
      b826 : Bool;
      b827 : Bool;
      b830 : Bool;
      b831 : Bool;
      b832 : Bool;
      b833 : Bool;
      b834 : Bool;
      b835 : Bool;
      b836 : Bool;
      b837 : Bool;
      b840 : Bool;
      b841 : Bool;
      b842 : Bool;
      b843 : Bool;
      b844 : Bool;
      b845 : Bool;
      b846 : Bool;
      b847 : Bool;
      b850 : Bool;
      b851 : Bool;
      b852 : Bool;
      b853 : Bool;
      b854 : Bool;
      b855 : Bool;
      b856 : Bool;
      b857 : Bool;
      b860 : Bool;
      b861 : Bool;
      b862 : Bool;
      b863 : Bool;
      b864 : Bool;
      b865 : Bool;
      b866 : Bool;
      b867 : Bool;
      b870 : Bool;
      b871 : Bool;
      b872 : Bool;
      b873 : Bool;
      b874 : Bool;
      b875 : Bool;
      b876 : Bool;
      b877 : Bool;
      b880 : Bool;
      b881 : Bool;
      b882 : Bool;
      b883 : Bool;
      b884 : Bool;
      b885 : Bool;
      b886 : Bool;
      b887 : Bool;
      b890 : Bool;
      b891 : Bool;
      b892 : Bool;
      b893 : Bool;
      b894 : Bool;
      b895 : Bool;
      b896 : Bool;
      b897 : Bool;
      b900 : Bool;
      b901 : Bool;
      b902 : Bool;
      b903 : Bool;
      b904 : Bool;
      b905 : Bool;
      b906 : Bool;
      b907 : Bool;
      b910 : Bool;
      b911 : Bool;
      b912 : Bool;
      b913 : Bool;
      b914 : Bool;
      b915 : Bool;
      b916 : Bool;
      b917 : Bool;
      b920 : Bool;
      b921 : Bool;
      b922 : Bool;
      b923 : Bool;
      b924 : Bool;
      b925 : Bool;
      b926 : Bool;
      b927 : Bool;
      b930 : Bool;
      b931 : Bool;
      b932 : Bool;
      b933 : Bool;
      b934 : Bool;
      b935 : Bool;
      b936 : Bool;
      b937 : Bool;
      b940 : Bool;
      b941 : Bool;
      b942 : Bool;
      b943 : Bool;
      b944 : Bool;
      b945 : Bool;
      b946 : Bool;
      b947 : Bool;
      b950 : Bool;
      b951 : Bool;
      b952 : Bool;
      b953 : Bool;
      b954 : Bool;
      b955 : Bool;
      b956 : Bool;
      b957 : Bool;
      b960 : Bool;
      b961 : Bool;
      b962 : Bool;
      b963 : Bool;
      b964 : Bool;
      b965 : Bool;
      b966 : Bool;
      b967 : Bool;
      b970 : Bool;
      b971 : Bool;
      b972 : Bool;
      b973 : Bool;
      b974 : Bool;
      b975 : Bool;
      b976 : Bool;
      b977 : Bool;
      b980 : Bool;
      b981 : Bool;
      b982 : Bool;
      b983 : Bool;
      b984 : Bool;
      b985 : Bool;
      b986 : Bool;
      b987 : Bool;
      b990 : Bool;
      b991 : Bool;
      b992 : Bool;
      b993 : Bool;
      b994 : Bool;
      b995 : Bool;
      b996 : Bool;
      b997 : Bool;
      b1000 : Bool;
      b1001 : Bool;
      b1002 : Bool;
      b1003 : Bool;
      b1004 : Bool;
      b1005 : Bool;
      b1006 : Bool;
      b1007 : Bool;
      b1010 : Bool;
      b1011 : Bool;
      b1012 : Bool;
      b1013 : Bool;
      b1014 : Bool;
      b1015 : Bool;
      b1016 : Bool;
      b1017 : Bool;
      b1020 : Bool;
      b1021 : Bool;
      b1022 : Bool;
      b1023 : Bool;
      b1024 : Bool;
      b1025 : Bool;
      b1026 : Bool;
      b1027 : Bool;
      b1030 : Bool;
      b1031 : Bool;
      b1032 : Bool;
      b1033 : Bool;
      b1034 : Bool;
      b1035 : Bool;
      b1036 : Bool;
      b1037 : Bool;
      b1040 : Bool;
      b1041 : Bool;
      b1042 : Bool;
      b1043 : Bool;
      b1044 : Bool;
      b1045 : Bool;
      b1046 : Bool;
      b1047 : Bool;
      b1050 : Bool;
      b1051 : Bool;
      b1052 : Bool;
      b1053 : Bool;
      b1054 : Bool;
      b1055 : Bool;
      b1056 : Bool;
      b1507 : Bool;
      b1060 : Bool;
      b1061 : Bool;
      b1062 : Bool;
      b1063 : Bool;
      b1064 : Bool;
      b1065 : Bool;
      b1066 : Bool;
      b1067 : Bool;
      b1070 : Bool;
      b1071 : Bool;
      b1072 : Bool;
      b1073 : Bool;
      b1074 : Bool;
      b1075 : Bool;
      b1076 : Bool;
      b1077 : Bool;
      b1080 : Bool;
      b1081 : Bool;
      b1082 : Bool;
      b1083 : Bool;
      b1084 : Bool;
      b1085 : Bool;
      b1086 : Bool;
      b1087 : Bool;
      b1090 : Bool;
      b1091 : Bool;
      b1092 : Bool;
      b1093 : Bool;
      b1094 : Bool;
      b1095 : Bool;
      b1096 : Bool;
      b1097 : Bool;
      b1100 : Bool;
      b1101 : Bool;
      b1102 : Bool;
      b1103 : Bool;
      b1104 : Bool;
      b1105 : Bool;
      b1106 : Bool;
      b1107 : Bool;
      b1110 : Bool;
      b1111 : Bool;
      b1112 : Bool;
      b1113 : Bool;
      b1114 : Bool;
      b1115 : Bool;
      b1116 : Bool;
      b1117 : Bool;
      b1120 : Bool;
      b1121 : Bool;
      b1122 : Bool;
      b1123 : Bool;
      b1124 : Bool;
      b1125 : Bool;
      b1126 : Bool;
      b1127 : Bool;
      b1130 : Bool;
      b1131 : Bool;
      b1132 : Bool;
      b1133 : Bool;
      b1134 : Bool;
      b1135 : Bool;
      b1136 : Bool;
      b1137 : Bool;
      b1140 : Bool;
      b1141 : Bool;
      b1142 : Bool;
      b1143 : Bool;
      b1144 : Bool;
      b1145 : Bool;
      b1146 : Bool;
      b1147 : Bool;
      b1150 : Bool;
      b1151 : Bool;
      b1152 : Bool;
      b1153 : Bool;
      b1154 : Bool;
      b1155 : Bool;
      b1156 : Bool;
      b1157 : Bool;
      b1160 : Bool;
      b1161 : Bool;
      b1162 : Bool;
      b1163 : Bool;
      b1164 : Bool;
      b1165 : Bool;
      b1166 : Bool;
      b1167 : Bool;
      b1170 : Bool;
      b1171 : Bool;
      b1172 : Bool;
      b1173 : Bool;
      b1174 : Bool;
      b1175 : Bool;
      b1176 : Bool;
      b1177 : Bool;
      b1180 : Bool;
      b1181 : Bool;
      b1182 : Bool;
      b1183 : Bool;
      b1184 : Bool;
      b1185 : Bool;
      b1186 : Bool;
      b1187 : Bool;
      b1190 : Bool;
      b1191 : Bool;
      b1192 : Bool;
      b1193 : Bool;
      b1194 : Bool;
      b1195 : Bool;
      b1196 : Bool;
      b1197 : Bool;
   END_STRUCT;


BEGIN

END_DATA_BLOCK

DATA_BLOCK "DB_FixWrite_Real"
{ S7_Optimized_Access := 'FALSE' }
VERSION : 0.0
   STRUCT
      R0 : Real;   // General.
      R4 : Real;
      R8 : Real;
      R12 : Real;
      R16 : Real;
      R20 : Real;
      R24 : Real;
      R28 : Real;
      R32 : Real;
      R36 : Real;
      R40 : Real;
      R44 : Real;
      R48 : Real;
      R52 : Real;
      R56 : Real;
      R60 : Real;
      R64 : Real;   // M501
      R68 : Real;
      R72 : Real;
      R76 : Real;
      R80 : Real;
      R84 : Real;
      R88 : Real;
      R92 : Real;
      R96 : Real;
      R100 : Real;
      R104 : Real;
      R108 : Real;
      R112 : Real;
      R116 : Real;
      R120 : Real;   // M502
      R124 : Real;
      R128 : Real;
      R132 : Real;
      R136 : Real;
      R140 : Real;
      R144 : Real;
      R148 : Real;
      R152 : Real;
      R156 : Real;
      R160 : Real;
      R164 : Real;
      R168 : Real;
      R172 : Real;
      R176 : Real;
      R180 : Real;   // M503.
      R184 : Real;
      R188 : Real;
      R192 : Real;
      R196 : Real;
      R200 : Real;
      R204 : Real;
      R208 : Real;
      R212 : Real;
      R216 : Real;
      R220 : Real;
      R224 : Real;
      R228 : Real;
      R232 : Real;
      R236 : Real;
      R240 : Real;   // M504
      R244 : Real;
      R248 : Real;
      R252 : Real;
      R256 : Real;
      R260 : Real;
      R264 : Real;
      R268 : Real;
      R272 : Real;
      R276 : Real;
      R280 : Real;
      R284 : Real;
      R288 : Real;
      R292 : Real;
      R296 : Real;
      R300 : Real;   // M505
      R304 : Real;
      R308 : Real;
      R312 : Real;
      R316 : Real;
      R320 : Real;
      R324 : Real;
      R328 : Real;
      R332 : Real;
      R336 : Real;
      R340 : Real;
      R344 : Real;
      R348 : Real;
      R352 : Real;
      R356 : Real;
      R360 : Real;   // M506 Spare value
      R364 : Real;   // M506.BQ3-left encoder min value (mm)
      R368 : Real;   // M506.BQ3-left encoder max value (mm)
      R372 : Real;   // M506.BQ4-right encoder min value (mm)
      R376 : Real;   // M506.BQ4-right encoder max value (mm)
      R380 : Real;
      R384 : Real;
      R388 : Real;
      R392 : Real;
      R396 : Real;
      R400 : Real;
      R404 : Real;
      R408 : Real;
      R412 : Real;
      R416 : Real;
      R420 : Real;
      R424 : Real;
      R428 : Real;
      R432 : Real;
      R436 : Real;
      R440 : Real;
      R444 : Real;
      R448 : Real;
      R452 : Real;
      R456 : Real;
      R460 : Real;
      R464 : Real;
      R468 : Real;
      R472 : Real;
      R476 : Real;
      R480 : Real;
      R484 : Real;
      R488 : Real;
      R492 : Real;
      R496 : Real;
   END_STRUCT;


BEGIN
   R104 := 6.0;
   R120 := 148.0;
   R124 := 35.0;
   R128 := 328.0;
   R132 := 35.0;
   R136 := 3.5;
   R140 := 355.0;
   R144 := 155.0;
   R148 := 175.0;
   R152 := 210.0;
   R156 := 335.0;
   R160 := 335.0;
   R164 := 355.0;
   R168 := 30.0;
   R172 := 100.0;
   R176 := 153.0;
   R180 := 213.0;
   R184 := 332.0;
   R188 := 33.0;
   R192 := 1.0;
   R196 := 6.0;
   R200 := 50.0;
   R208 := 1179.0;
   R216 := 1.0;
   R220 := 6.0;
   R224 := 50.0;
   R232 := 955.0;
   R300 := 2.0;
   R304 := 6.0;
   R308 := 50.0;
   R316 := 2244.0;
   R320 := -138.2032;
   R360 := 1.0;
   R364 := 885.0;
   R368 := 2012.0;
   R372 := 870.0;
   R376 := 2006.0;

END_DATA_BLOCK

DATA_BLOCK "DB_FixWriteDint"
{ S7_Optimized_Access := 'FALSE' }
VERSION : 0.0
   STRUCT
      DW0 : DInt;   // General.
      DW4 : DInt;
      DW8 : DInt;
      DW12 : DInt;
      DW16 : DInt;
      DW20 : DInt;
      DW24 : DInt;
      DW28 : DInt;
      DW32 : DInt;
      DW36 : DInt;
      DW40 : DInt;
      DW44 : DInt;
      DW48 : DInt;
      DW52 : DInt;
      DW56 : DInt;
      DW60 : DInt;   // M501
      DW64 : DInt;   // M501
      DW68 : DInt;
      DW72 : DInt;
      DW76 : DInt;
      DW80 : DInt;
      DW84 : DInt;
      DW88 : DInt;
      DW92 : DInt;
      DW96 : DInt;
      DW100 : DInt;
      DW104 : DInt;
      DW108 : DInt;
      DW112 : DInt;
      DW116 : DInt;
      DW120 : DInt;   // M502
      DW124 : DInt;
      DW128 : DInt;
      DW132 : DInt;
      DW136 : DInt;
      DW140 : DInt;
      DW144 : DInt;
      DW148 : DInt;
      DW152 : DInt;
      DW156 : DInt;
      DW160 : DInt;
      DW164 : DInt;
      DW168 : DInt;
      DW172 : DInt;
      DW176 : DInt;
      DW180 : DInt;   // M503. Preset on rotator encoder [pulses]
      DW184 : DInt;   // M503 Stop starting position lower limit (imp)
      DW188 : DInt;   // M503 Stop starting position upper limit (imp)
      DW192 : DInt;   // M503 Slowdown end position lower limit (imp)
      DW196 : DInt;   // M503 Slowdown end position upper limit (imp)
      DW200 : DInt;   // M503 Stop end position lower limit (imp)
      DW204 : DInt;   // M503 Stop end position upper limit (imp)
      DW208 : DInt;
      DW212 : DInt;
      DW216 : DInt;
      DW220 : DInt;
      DW224 : DInt;
      DW228 : DInt;
      DW232 : DInt;
      DW236 : DInt;
      DW240 : DInt;   // M504
      DW244 : DInt;
      DW248 : DInt;
      DW252 : DInt;
      DW256 : DInt;
      DW260 : DInt;
      DW264 : DInt;
      DW268 : DInt;
      DW272 : DInt;
      DW276 : DInt;
      DW280 : DInt;
      DW284 : DInt;
      DW288 : DInt;
      DW292 : DInt;
      DW296 : DInt;
      DW300 : DInt;   // M505
      DW304 : DInt;
      DW308 : DInt;
      DW312 : DInt;
      DW316 : DInt;
      DW320 : DInt;
      DW324 : DInt;
      DW328 : DInt;
      DW332 : DInt;
      DW336 : DInt;
      DW340 : DInt;
      DW344 : DInt;
      DW348 : DInt;
      DW352 : DInt;
      DW356 : DInt;
      DW360 : DInt;   // M506. Preset on left side MLD encoder [pulses]
      DW364 : DInt;   // M506. Preset on right side MLD encoder [pulses]
      DW368 : DInt;
      DW372 : DInt;
      DW376 : DInt;
      DW380 : DInt;
      DW384 : DInt;
      DW388 : DInt;
      DW392 : DInt;
      DW396 : DInt;
      DW400 : DInt;
      DW404 : DInt;
      DW408 : DInt;
      DW412 : DInt;
      DW416 : DInt;
      DW420 : DInt;
      DW424 : DInt;
      DW428 : DInt;
      DW432 : DInt;
      DW436 : DInt;
      DW440 : DInt;
      DW444 : DInt;
      DW448 : DInt;
      DW452 : DInt;
      DW456 : DInt;
      DW460 : DInt;
      DW464 : DInt;
      DW468 : DInt;
      DW472 : DInt;
      DW476 : DInt;
      DW480 : DInt;
      DW484 : DInt;
      DW488 : DInt;
      DW492 : DInt;
      DW496 : DInt;
      DW500 : DInt;
      DW504 : DInt;
      DW508 : DInt;
      DW512 : DInt;
      DW516 : DInt;
      DW520 : DInt;
      DW524 : DInt;
      DW528 : DInt;
      DW532 : DInt;
      DW536 : DInt;
      DW540 : DInt;
      DW544 : DInt;
      DW548 : DInt;
      DW552 : DInt;
      DW556 : DInt;
      DW560 : DInt;
      DW564 : DInt;
      DW568 : DInt;
      DW572 : DInt;
      DW576 : DInt;
      DW580 : DInt;
      DW584 : DInt;
      DW588 : DInt;
      DW592 : DInt;
      DW596 : DInt;
      DW600 : DInt;
      DW604 : DInt;
      DW608 : DInt;
      DW612 : DInt;
      DW616 : DInt;
      DW620 : DInt;
      DW624 : DInt;
      DW628 : DInt;
      DW632 : DInt;
      DW636 : DInt;
      DW640 : DInt;
      DW644 : DInt;
      DW648 : DInt;
      DW652 : DInt;
      DW656 : DInt;
      DW660 : DInt;
      DW664 : DInt;
      DW668 : DInt;
      DW672 : DInt;
      DW676 : DInt;
      DW680 : DInt;
      DW684 : DInt;
      DW688 : DInt;
      DW692 : DInt;
      DW696 : DInt;
      DW700 : DInt;
      DW704 : DInt;
      DW708 : DInt;
      DW712 : DInt;
      DW716 : DInt;
      DW720 : DInt;
      DW724 : DInt;
      DW728 : DInt;
      DW732 : DInt;
      DW736 : DInt;
      DW740 : DInt;
      DW744 : DInt;
      DW748 : DInt;
      DW752 : DInt;
      DW756 : DInt;
      DW760 : DInt;
      DW764 : DInt;
      DW768 : DInt;
      DW772 : DInt;
      DW776 : DInt;
      DW780 : DInt;
      DW784 : DInt;
      DW788 : DInt;
      DW792 : DInt;
      DW796 : DInt;
      DW800 : DInt;
      DW804 : DInt;
      DW808 : DInt;
      DW812 : DInt;
      DW816 : DInt;
      DW820 : DInt;
      DW824 : DInt;
      DW828 : DInt;
      DW832 : DInt;
      DW836 : DInt;
      DW840 : DInt;
      DW844 : DInt;
      DW848 : DInt;
      DW852 : DInt;
      DW856 : DInt;
      DW860 : DInt;
      DW864 : DInt;
      DW868 : DInt;
      DW872 : DInt;
      DW876 : DInt;
      DW880 : DInt;
      DW884 : DInt;
      DW888 : DInt;
      DW892 : DInt;
      DW896 : DInt;
   END_STRUCT;


BEGIN
   DW128 := DINT#100000;
   DW184 := DINT#-10;
   DW188 := DINT#10000;
   DW192 := DINT#325000;
   DW196 := DINT#495000;
   DW200 := DINT#416000;
   DW204 := DINT#435000;
   DW300 := DINT#100000;
   DW360 := DINT#10000;
   DW364 := DINT#10000;
   DW380 := DINT#2300;
   DW384 := DINT#2300;
   DW392 := DINT#4600;
   DW404 := DINT#3210;
   DW428 := DINT#1605;
   DW432 := DINT#1605;
   DW520 := DINT#1527177;
   DW532 := DINT#252366;
   DW536 := DINT#91114;

END_DATA_BLOCK

DATA_BLOCK "DB_FixWriteInt"
{ S7_Optimized_Access := 'FALSE' }
VERSION : 0.1
   STRUCT
      W0 : Int;
      W2 : Int;
      W4 : Int;
      W6 : Int;
      W8 : Int;
      W10 : Int;   // Z500.Automatic speed selection (1=20;3=40 4=60 5=80) m/min
      W12 : Int;
      W14 : Int;   // Z500.Manual speed selection (1=20;3=40 4=60 5=80) m/min
      W16 : Int;
      W18 : Int;   // Z500. Line Enable (1=enable 0=no )
      W20 : Int;
      W22 : Int;
      W24 : Int;   // Z500.Selection conveyor start clean (M501-M506) (requested)
      W26 : Int;
      W28 : Int;
      BitNuovi : Struct   // struct created to use this word, relative to "Portrait=1 /Landscape=2" as a bit
         byteMSD : Byte;
         bit0 : Bool;   // Z500.Selection Unloading mode =Portrait
         bit1 : Bool;   // Z500.Selection Unloading mode =Landescape
      END_STRUCT;
      W32 : Int;
      W34 : Int;
      W36 : Int;
      W38 : Int;
      W40 : Int;
      W42 : Int;
      W44 : Int;
      W46 : Int;
      W48 : Int;
      W50 : Int;   // M501
      W52 : Int;   // M501. Distance from phot.B1..B1D to middle of conv.(section Z1/Z2) (MLD) [mm]
      W54 : Int;   // M501. Offset positioning on tail - on conveyor section Z1(MLD) [mm] -/+
      W56 : Int;
      W58 : Int;   // M501. Distance from phot.B1..B1D to end of the conveyor section Z2 (MLD) [mm]
      W60 : Int;   // M501. Offset positioning on tail -  conveyor section Z2 (MLD) [mm] -/+
      W62 : Int;
      W64 : Int;   // M501. Offset positioning on middle of conveyor (section Z1/Z2) (MLD) [mm] -/+
      W66 : Int;
      W68 : Int;
      W70 : Int;   // M502
      W72 : Int;   // M502. Distance from phot.M502 B1B2 to center of Rotator M503 (LLD) [mm]
      W74 : Int;   // M502 Offset positioning on center of Rotator (LLD) [mm]-/+
      W76 : Int;   // M502. Distance from phot.M502 B1B2 to end of conveyor (LLD)[mm]
      W78 : Int;   // M502 Offset positioning on end of conveyor [mm] (LLD)-/+
      W80 : Int;
      W82 : Int;
      W84 : Int;
      W86 : Int;
      W88 : Int;
      M502_DIST_FTC : Int;   // M503
      M502_OFFST_SQR : Int;
      W94 : Int;
      W96 : Int;
      M502_M1_OFFST_STOP_END : Int;
      M502_M2_OFFST_STOP_BEG : Int;
      M502_M2_OFFST_STOP_END : Int;
      M502_DIST_CAPS : Int;
      W106 : Int;
      W108 : Int;
      W110 : Int;   // M504.spare word 1
      W112 : Int;   // M504.spare word 2
      W114 : Int;
      W116 : Int;   // M504 Speed reduction during unpacking (0= OFF 1= ON)
      W118 : Int;   // M504 Move Backward enable status (0= OFF 1= ON)
      W120 : Int;
      W122 : Int;
      W124 : Int;
      W126 : Int;
      W128 : Int;
      W130 : Int;   // M505.spare word 1
      W132 : Int;   // M505.spare word 2
      W134 : Int;   // M505.Time of squaring (s/100)
      W136 : Int;   // M505 squaring speed of rotation (mt/min)
      W138 : Int;   // M505.Offset space to adjust M505 slowdown position Mono (mm)
      W140 : Int;
      W142 : Int;
      W144 : Int;
      W146 : Int;
      W148 : Int;
      M506_B_OffsetLLD : Int;   // M506.Offset space to adjust M506Left position (LLD)(mm)-/+
      M506_Mono_OffsetLLD : Int;   // M506.Offset space to adjust M506centered position (LLD)(mm)-/+
      M506_A_OffsetLLD : Int;   // M506.Offset space to adjust M506Right position (LLD)(mm)-/+
      W156 : Int;   // M506. Distance between 2 Lite when squared (MLD)(do not use)[mm]
      W158 : Int;   // M506. Lateral offset on sheets Side A (Stereo) (MLD)[mm] -/+
      W160 : Int;   // M506. Lateral offset on sheets Side B (Stereo) (MLD)[mm] -/+
      W162 : Int;   // M506. Lateral offset on sheets MONO (MLD)[mm] -/+
      W164 : Int;
      W166 : Int;   // M506 high lateral speed of rotation MLD (mt/min)
      W168 : Int;   // M506 low lateral speed of rotation MLD (mt/min)
      W170 : Int;   // M506. Spare word 02 (MLD)[mm]
      W172 : Int;   // M506. Spare word 03 (LLD)[mm]
      W174 : Int;
      W176 : Int;
      W178 : Int;
      W180 : Int;
      W182 : Int;
      W184 : Int;
      W186 : Int;
      W188 : Int;
      W190 : Int;
      W192 : Int;
      W194 : Int;
      W196 : Int;
      W198 : Int;
      W200 : Int;
      W202 : Int;
      W204 : Int;
      W206 : Int;
      W208 : Int;
      W210 : Int;
      W212 : Int;
      W214 : Int;
      W216 : Int;
      W218 : Int;
      W220 : Int;
      W222 : Int;
      W224 : Int;
      W226 : Int;
      W228 : Int;
      W230 : Int;
      W232 : Int;
      W234 : Int;
      W236 : Int;
      W238 : Int;
      W240 : Int;
      W242 : Int;
      W244 : Int;
      W246 : Int;
      W248 : Int;
      W250 : Int;
      W252 : Int;
      W254 : Int;
      W256 : Int;
      W258 : Int;
      W260 : Int;
      W262 : Int;
      W264 : Int;
      W266 : Int;
      W268 : Int;
      W270 : Int;
      W272 : Int;
      W274 : Int;
      W276 : Int;
      W278 : Int;
      W280 : Int;
      W282 : Int;
      W284 : Int;
      W286 : Int;
      W288 : Int;
      W290 : Int;
      W292 : Int;
      W294 : Int;
      W296 : Int;
      W298 : Int;
      W300 : Int;   // LES1_M507: (0= DISABLED  1= ENABLE)
      W302 : Int;
      W304 : Int;
      W306 : Int;
      W308 : Int;
      W310 : Int;
      W312 : Int;
      W314 : Int;
      W316 : Int;
      W318 : Int;
      W320 : Int;
      W322 : Int;
      W324 : Int;
      W326 : Int;
      W328 : Int;
      W330 : Int;
      W332 : Int;
      W334 : Int;
      W336 : Int;
      W338 : Int;
      W340 : Int;
      W342 : Int;
      W344 : Int;
      W346 : Int;
      W348 : Int;
      W350 : Int;
      W352 : Int;
      W354 : Int;
      W356 : Int;
      W358 : Int;
      W360 : Int;
      W362 : Int;
      W364 : Int;
      W366 : Int;
      W368 : Int;
      W370 : Int;
      W372 : Int;
      W374 : Int;
      W376 : Int;
      W378 : Int;
      W380 : Int;
      W382 : Int;
      W384 : Int;
      W386 : Int;
      W388 : Int;
      W390 : Int;
      W392 : Int;
      W394 : Int;
      W396 : Int;
      W398 : Int;
      W400 : Int;
      W402 : Int;
      W404 : Int;
      W406 : Int;
      W408 : Int;
      W410 : Int;
      W412 : Int;
      W414 : Int;
      W416 : Int;
      W418 : Int;
      W420 : Int;
      W422 : Int;
      W424 : Int;
      W426 : Int;
      W428 : Int;
      W430 : Int;
      W432 : Int;
      W434 : Int;
      W436 : Int;
      W438 : Int;
      W440 : Int;
      W442 : Int;
      W444 : Int;
      W446 : Int;
      W448 : Int;
      W450 : Int;
      W452 : Int;
      W454 : Int;
      W456 : Int;
      W458 : Int;
      W460 : Int;
      W462 : Int;
      W464 : Int;
      W466 : Int;
      W468 : Int;
      W470 : Int;
      W472 : Int;
      W474 : Int;
      W476 : Int;
      W478 : Int;
      W480 : Int;
      W482 : Int;
      W484 : Int;
      W486 : Int;
      W488 : Int;
      W490 : Int;
      W492 : Int;
      W494 : Int;
      W496 : Int;
      W498 : Int;
      W500 : Int;
      W502 : Int;
      W504 : Int;
      W506 : Int;
      W508 : Int;
      W510 : Int;
      W512 : Int;
      W514 : Int;
      W516 : Int;
      W518 : Int;
      W520 : Int;
      W522 : Int;
      W524 : Int;
      W526 : Int;
      W528 : Int;
      W530 : Int;
      W532 : Int;
      W534 : Int;
      W536 : Int;
      W538 : Int;
      W540 : Int;
      W542 : Int;
      W544 : Int;
      W546 : Int;
      W548 : Int;
      W550 : Int;
      W552 : Int;
      W554 : Int;
      W556 : Int;
      W558 : Int;
      W560 : Int;
      W562 : Int;
      W564 : Int;
      W566 : Int;
      W568 : Int;
      W570 : Int;
      W572 : Int;
      W574 : Int;
      W576 : Int;
      W578 : Int;
      W580 : Int;
      W582 : Int;
      W584 : Int;
      W586 : Int;
      W588 : Int;
      W590 : Int;
      W592 : Int;
      W594 : Int;
      W596 : Int;
      W598 : Int;
   END_STRUCT;


BEGIN
   W10 := 4;
   W14 := 1;
   W16 := 5;
   W18 := 1;
   W24 := 506;
   W26 := 505;
   W52 := 2720;
   W58 := 4670;
   W72 := 2100;
   W74 := 75;
   W76 := 4100;
   M502_DIST_FTC := 600;
   M502_OFFST_SQR := -130;
   M502_M1_OFFST_STOP_END := -90;
   M502_M2_OFFST_STOP_END := -390;
   M502_DIST_CAPS := 50;
   W106 := 150;
   W108 := 150;
   W118 := 1;
   W120 := 400;
   W122 := 270;
   W124 := 305;
   W126 := 635;
   W128 := 305;
   W134 := 300;
   W136 := 6;
   W138 := 620;
   W140 := 620;
   W142 := 400;
   W144 := 270;
   W148 := 20;
   M506_Mono_OffsetLLD := 35;
   W156 := 5;
   W162 := -15;
   W164 := 15;
   W166 := 30;
   W168 := 7;
   W174 := 200;
   W176 := 10;
   W178 := 3;
   W190 := 400;
   W192 := 150;
   W194 := 200;
   W196 := 10;
   W198 := 3;
   W210 := 2770;
   W214 := 1;
   W216 := 2;
   W218 := 2750;
   W220 := 500;
   W222 := 460;
   W224 := 630;
   W226 := 1110;
   W230 := 965;
   W232 := 100;
   W234 := 50;
   W250 := 2934;
   W252 := 169;
   W256 := -45;
   W260 := 30;
   W270 := 400;
   W272 := 150;
   W274 := 150;
   W276 := 10;
   W278 := 10;
   W402 := 10;

END_DATA_BLOCK

DATA_BLOCK "DB_Fix write bit"
{ S7_Optimized_Access := 'FALSE' }
VERSION : 0.0
   STRUCT
      b00 : Bool;   // Z500. Manual mode request
      b01 : Bool;   // Z500. Automatic mode request
      b02 : Bool;   // Z500. Clean zone request
      b03 : Bool;   // Z500. Stop clean zone request
      b04 : Bool;
      b05 : Bool;   // Z500.Start cycle
      b06 : Bool;   // Z500.Stop cycle
      b07 : Bool;   // Z500.Reset Request of all the conveyors
      b10 : Bool;   // Z500.Reset anomaly
      b11 : Bool;
      b12 : Bool;
      b13 : Bool;
      b14 : Bool;
      b15 : Bool;
      b16 : Bool;
      b17 : Bool;
      b20 : Bool;
      b21 : Bool;
      b22 : Bool;   // Z500.Active mono mode forcing
      b23 : Bool;   // Z500.Disactive mono mode forcing
      b24 : Bool;
      b25 : Bool;
      b26 : Bool;
      b27 : Bool;
      b30 : Bool;
      b31 : Bool;
      b32 : Bool;
      b33 : Bool;
      b34 : Bool;
      b35 : Bool;
      b36 : Bool;
      b37 : Bool;
      b40 : Bool;   // M501
      b41 : Bool;
      b42 : Bool;   // M501 Clean P.Button forward in MLD  M1 M2 M3 (Z0 Z1 Z2)
      b43 : Bool;   // M501 Clean P.Button forward in MLD M2 M3 (Z1 Z2)
      b44 : Bool;   // M501 Clean P.Button Backward in MLD M2 M3 (Z1 Z2)
      b45 : Bool;
      b46 : Bool;
      b47 : Bool;   // M501 Reset Request
      b50 : Bool;
      b51 : Bool;   // M501 Z1-Z2 Unload P.B
      b52 : Bool;   // M501 Line activation On/OFF P.B.
      b53 : Bool;
      b54 : Bool;
      b55 : Bool;
      b56 : Bool;
      b57 : Bool;
      b60 : Bool;   // M502
      b61 : Bool;
      b62 : Bool;
      b63 : Bool;
      b64 : Bool;
      b65 : Bool;
      b66 : Bool;
      FIX_RESET_REQ_M502 : Bool;   // M502 Reset Request
      b70 : Bool;
      b71 : Bool;
      b72 : Bool;
      b73 : Bool;
      b74 : Bool;
      b75 : Bool;
      b76 : Bool;
      b77 : Bool;
      b80 : Bool;   // M503 Preset encoder of Rotator frame
      b81 : Bool;
      b82 : Bool;
      b83 : Bool;
      b84 : Bool;
      b85 : Bool;
      b86 : Bool;
      FIX_RESET_REQ_M503 : Bool;   // M503 Reset Request
      b90 : Bool;
      b91 : Bool;
      b92 : Bool;
      b93 : Bool;
      b94 : Bool;
      b95 : Bool;
      b96 : Bool;
      b97 : Bool;
      b100 : Bool;   // M504
      b101 : Bool;
      b102 : Bool;
      b103 : Bool;
      b104 : Bool;
      b105 : Bool;
      b106 : Bool;
      FIX_RESET_REQ_M504 : Bool;   // M504 Reset Request
      b110 : Bool;
      b111 : Bool;
      b112 : Bool;
      b113 : Bool;
      b114 : Bool;
      b115 : Bool;
      b116 : Bool;
      b117 : Bool;
      b120 : Bool;   // M505
      b121 : Bool;
      b122 : Bool;
      b123 : Bool;
      b124 : Bool;
      b125 : Bool;
      b126 : Bool;
      FIX_RESET_REQ_M505 : Bool;   // M505 Reset Request
      b130 : Bool;
      b131 : Bool;
      b132 : Bool;
      b133 : Bool;
      b134 : Bool;
      b135 : Bool;
      b136 : Bool;
      b137 : Bool;
      b140 : Bool;   // M506. Preset Encoder of Right Side
      b141 : Bool;   // M506. Preset Encoder on Left Side
      b142 : Bool;   // M506. Calibration Min Value  Encoder Right Side
      b143 : Bool;   // M506. Calibration Max Value Encoder Right Side
      b144 : Bool;   // M506. Calibration Min Value  Encoder Left Side
      b145 : Bool;   // M506. Calibration Max Value Encoder Left Side
      b146 : Bool;
      FIX_RESET_REQ_M506 : Bool;   // M506 Reset Request
      b150 : Bool;   // M506 glass step forward LLD
      b151 : Bool;   // M506 Request to Reposition Photocells
      b152 : Bool;   // M506 glass step backward LLD
      b153 : Bool;   // M506 glass Squaring repetition MLD
      b154 : Bool;
      b155 : Bool;
      b156 : Bool;
      b157 : Bool;
      b160 : Bool;
      b161 : Bool;
      b162 : Bool;
      b163 : Bool;
      b164 : Bool;
      b165 : Bool;
      b166 : Bool;
      b167 : Bool;
      b170 : Bool;
      b171 : Bool;
      b172 : Bool;
      b173 : Bool;
      b174 : Bool;
      b175 : Bool;
      b176 : Bool;
      b177 : Bool;
      b180 : Bool;
      b181 : Bool;
      b182 : Bool;
      b183 : Bool;
      b184 : Bool;
      b185 : Bool;
      b186 : Bool;
      b187 : Bool;
      b190 : Bool;
      b191 : Bool;
      b192 : Bool;
      b193 : Bool;
      b194 : Bool;
      b195 : Bool;
      b196 : Bool;
      b197 : Bool;
      b200 : Bool;
      b201 : Bool;
      b202 : Bool;
      b203 : Bool;
      b204 : Bool;
      b205 : Bool;
      b206 : Bool;
      b207 : Bool;
      b210 : Bool;
      b211 : Bool;
      b212 : Bool;
      b213 : Bool;
      b214 : Bool;
      b215 : Bool;
      b216 : Bool;
      b217 : Bool;
      b220 : Bool;
      b221 : Bool;
      b222 : Bool;
      b223 : Bool;
      b224 : Bool;
      b225 : Bool;
      b226 : Bool;
      b227 : Bool;
      b230 : Bool;
      b231 : Bool;
      b232 : Bool;
      b233 : Bool;
      b234 : Bool;
      b235 : Bool;
      b236 : Bool;
      b237 : Bool;
      b240 : Bool;
      b241 : Bool;
      b242 : Bool;
      b243 : Bool;
      b244 : Bool;
      b245 : Bool;
      b246 : Bool;
      b247 : Bool;
      b250 : Bool;
      b251 : Bool;
      b252 : Bool;
      b253 : Bool;
      b254 : Bool;
      b255 : Bool;
      b256 : Bool;
      b257 : Bool;
      b260 : Bool;
      b261 : Bool;
      b262 : Bool;
      b263 : Bool;
      b264 : Bool;
      b265 : Bool;
      b266 : Bool;
      b267 : Bool;
      b270 : Bool;
      b271 : Bool;
      b272 : Bool;
      b273 : Bool;
      b274 : Bool;
      b275 : Bool;
      b276 : Bool;
      b277 : Bool;
      b280 : Bool;   // M508.
      b281 : Bool;
      b282 : Bool;
      b283 : Bool;
      b284 : Bool;
      b285 : Bool;
      b286 : Bool;
      b287 : Bool;
      b290 : Bool;
      b291 : Bool;
      b292 : Bool;
      b293 : Bool;
      b294 : Bool;
      b295 : Bool;
      b296 : Bool;
      b297 : Bool;
      b300 : Bool;   // M509. Preset Encoder on Squaring Request
      b301 : Bool;   // M509. Calibration Min Value Squaring Encoder
      b302 : Bool;   // M509. Calibration Max Value Squaring Encoder
      b303 : Bool;
      b304 : Bool;
      b305 : Bool;
      b306 : Bool;
      b307 : Bool;
      b310 : Bool;
      b311 : Bool;
      b312 : Bool;
      b313 : Bool;
      b314 : Bool;
      b315 : Bool;
      b316 : Bool;
      b317 : Bool;
      b320 : Bool;
      b321 : Bool;
      b322 : Bool;
      b323 : Bool;
      b324 : Bool;
      b325 : Bool;
      b326 : Bool;
      b327 : Bool;
      b330 : Bool;
      b331 : Bool;
      b332 : Bool;
      b333 : Bool;
      b334 : Bool;
      b335 : Bool;
      b336 : Bool;
      b337 : Bool;
      b340 : Bool;
      b341 : Bool;
      b342 : Bool;
      b343 : Bool;
      b344 : Bool;
      b345 : Bool;
      b346 : Bool;
      b347 : Bool;
      b350 : Bool;
      b351 : Bool;
      b352 : Bool;
      b353 : Bool;
      b354 : Bool;
      b355 : Bool;
      b356 : Bool;
      b357 : Bool;
      b360 : Bool;
      b361 : Bool;
      b362 : Bool;
      b363 : Bool;
      b364 : Bool;
      b365 : Bool;
      b366 : Bool;
      b367 : Bool;
      b370 : Bool;
      b371 : Bool;
      b372 : Bool;
      b373 : Bool;
      b374 : Bool;
      b375 : Bool;
      b376 : Bool;
      b377 : Bool;
      b380 : Bool;
      b381 : Bool;
      b382 : Bool;
      b383 : Bool;
      b384 : Bool;
      b385 : Bool;
      b386 : Bool;
      b387 : Bool;
      b390 : Bool;
      b391 : Bool;
      b392 : Bool;
      b393 : Bool;
      b394 : Bool;
      b395 : Bool;
      b396 : Bool;
      b397 : Bool;
      b400 : Bool;   // M510. Start Cycle
      b401 : Bool;   // M510. Stop Cycle
      b402 : Bool;
      b403 : Bool;
      b404 : Bool;
      b405 : Bool;
      b406 : Bool;
      b407 : Bool;
      b410 : Bool;
      b411 : Bool;
      b412 : Bool;
      b413 : Bool;
      b414 : Bool;
      b415 : Bool;
      b416 : Bool;
      b417 : Bool;
      b420 : Bool;
      b421 : Bool;
      b422 : Bool;
      b423 : Bool;
      b424 : Bool;
      b425 : Bool;
      b426 : Bool;
      b427 : Bool;
      b430 : Bool;
      b431 : Bool;
      b432 : Bool;
      b433 : Bool;
      b434 : Bool;
      b435 : Bool;
      b436 : Bool;
      b437 : Bool;
      b440 : Bool;
      b441 : Bool;
      b442 : Bool;
      b443 : Bool;
      b444 : Bool;
      b445 : Bool;
      b446 : Bool;
      b447 : Bool;
      b450 : Bool;
      b451 : Bool;
      b452 : Bool;
      b453 : Bool;
      b454 : Bool;
      b455 : Bool;
      b456 : Bool;
      b457 : Bool;
      b460 : Bool;
      b461 : Bool;
      b462 : Bool;
      b463 : Bool;
      b464 : Bool;
      b465 : Bool;
      b466 : Bool;
      b467 : Bool;
      b470 : Bool;
      b471 : Bool;
      b472 : Bool;
      b473 : Bool;
      b474 : Bool;
      b475 : Bool;
      b476 : Bool;
      b477 : Bool;
      b480 : Bool;
      b481 : Bool;
      b482 : Bool;
      b483 : Bool;
      b484 : Bool;
      b485 : Bool;
      b486 : Bool;
      b487 : Bool;
      b490 : Bool;
      b491 : Bool;
      b492 : Bool;
      b493 : Bool;
      b494 : Bool;
      b495 : Bool;
      b496 : Bool;
      b497 : Bool;
      b500 : Bool;
      b501 : Bool;
      b502 : Bool;
      b503 : Bool;
      b504 : Bool;
      b505 : Bool;
      b506 : Bool;
      b507 : Bool;
      b510 : Bool;
      b511 : Bool;
      b512 : Bool;
      b513 : Bool;
      b514 : Bool;
      b515 : Bool;
      b516 : Bool;
      b517 : Bool;
      b520 : Bool;
      b521 : Bool;
      b522 : Bool;
      b523 : Bool;
      b524 : Bool;
      b525 : Bool;
      b526 : Bool;
      b527 : Bool;
      b530 : Bool;
      b531 : Bool;
      b532 : Bool;
      b533 : Bool;
      b534 : Bool;
      b535 : Bool;
      b536 : Bool;
      b537 : Bool;
      b540 : Bool;
      b541 : Bool;
      b542 : Bool;
      b543 : Bool;
      b544 : Bool;
      b545 : Bool;
      b546 : Bool;
      b547 : Bool;
      b550 : Bool;
      b551 : Bool;
      b552 : Bool;
      b553 : Bool;
      b554 : Bool;
      b555 : Bool;
      b556 : Bool;
      b557 : Bool;
      b560 : Bool;
      b561 : Bool;
      b562 : Bool;
      b563 : Bool;
      b564 : Bool;
      b565 : Bool;
      b566 : Bool;
      b567 : Bool;
      b570 : Bool;
      b571 : Bool;
      b572 : Bool;
      b573 : Bool;
      b574 : Bool;
      b575 : Bool;
      b576 : Bool;
      b577 : Bool;
      b580 : Bool;
      b581 : Bool;
      b582 : Bool;
      b583 : Bool;
      b584 : Bool;
      b585 : Bool;
      b586 : Bool;
      b587 : Bool;
      b590 : Bool;
      b591 : Bool;
      b592 : Bool;
      b593 : Bool;
      b594 : Bool;
      b595 : Bool;
      b596 : Bool;
      b597 : Bool;
      b600 : Bool;
      b601 : Bool;
      b602 : Bool;
      b603 : Bool;
      b604 : Bool;
      b605 : Bool;
      b606 : Bool;
      b607 : Bool;
      b610 : Bool;
      b611 : Bool;
      b612 : Bool;
      b613 : Bool;
      b614 : Bool;
      b615 : Bool;
      b616 : Bool;
      b617 : Bool;
      b620 : Bool;
      b621 : Bool;
      b622 : Bool;
      b623 : Bool;
      b624 : Bool;
      b625 : Bool;
      b626 : Bool;
      b627 : Bool;
      b630 : Bool;
      b631 : Bool;
      b632 : Bool;
      b633 : Bool;
      b634 : Bool;
      b635 : Bool;
      b636 : Bool;
      b637 : Bool;
      b640 : Bool;
      b641 : Bool;
      b642 : Bool;
      b643 : Bool;
      b644 : Bool;
      b645 : Bool;
      b646 : Bool;
      b647 : Bool;
      b650 : Bool;
      b651 : Bool;
      b652 : Bool;
      b653 : Bool;
      b654 : Bool;
      b655 : Bool;
      b656 : Bool;
      b657 : Bool;
      b660 : Bool;
      b661 : Bool;
      b662 : Bool;
      b663 : Bool;
      b664 : Bool;
      b665 : Bool;
      b666 : Bool;
      b667 : Bool;
      b670 : Bool;
      b671 : Bool;
      b672 : Bool;
      b673 : Bool;
      b674 : Bool;
      b675 : Bool;
      b676 : Bool;
      b677 : Bool;
      b680 : Bool;
      b681 : Bool;
      b682 : Bool;
      b683 : Bool;
      b684 : Bool;
      b685 : Bool;
      b686 : Bool;
      b687 : Bool;
      b690 : Bool;
      b691 : Bool;
      b692 : Bool;
      b693 : Bool;
      b694 : Bool;
      b695 : Bool;
      b696 : Bool;
      b697 : Bool;
      b700 : Bool;
      b701 : Bool;
      b702 : Bool;
      b703 : Bool;
      b704 : Bool;
      b705 : Bool;
      b706 : Bool;
      b707 : Bool;
      b710 : Bool;
      b711 : Bool;
      b712 : Bool;
      b713 : Bool;
      b714 : Bool;
      b715 : Bool;
      b716 : Bool;
      b717 : Bool;
      b720 : Bool;
      b721 : Bool;
      b722 : Bool;
      b723 : Bool;
      b724 : Bool;
      b725 : Bool;
      b726 : Bool;
      b727 : Bool;
      b730 : Bool;
      b731 : Bool;
      b732 : Bool;
      b733 : Bool;
      b734 : Bool;
      b735 : Bool;
      b736 : Bool;
      b737 : Bool;
      b740 : Bool;
      b741 : Bool;
      b742 : Bool;
      b743 : Bool;
      b744 : Bool;
      b745 : Bool;
      b746 : Bool;
      b747 : Bool;
      b750 : Bool;
      b751 : Bool;
      b752 : Bool;
      b753 : Bool;
      b754 : Bool;
      b755 : Bool;
      b756 : Bool;
      b757 : Bool;
      b760 : Bool;
      b761 : Bool;
      b762 : Bool;
      b763 : Bool;
      b764 : Bool;
      b765 : Bool;
      b766 : Bool;
      b767 : Bool;
      b770 : Bool;
      b771 : Bool;
      b772 : Bool;
      b773 : Bool;
      b774 : Bool;
      b775 : Bool;
      b776 : Bool;
      b777 : Bool;
      b780 : Bool;
      b781 : Bool;
      b782 : Bool;
      b783 : Bool;
      b784 : Bool;
      b785 : Bool;
      b786 : Bool;
      b787 : Bool;
      b790 : Bool;
      b791 : Bool;
      b792 : Bool;
      b793 : Bool;
      b794 : Bool;
      b795 : Bool;
      b796 : Bool;
      b797 : Bool;
      b800 : Bool;
      b801 : Bool;
      b802 : Bool;
      b803 : Bool;
      b804 : Bool;
      b805 : Bool;
      b806 : Bool;
      b807 : Bool;
      b810 : Bool;
      b811 : Bool;
      b812 : Bool;
      b813 : Bool;
      b814 : Bool;
      b815 : Bool;
      b816 : Bool;
      b817 : Bool;
      b820 : Bool;
      b821 : Bool;
      b822 : Bool;
      b823 : Bool;
      b824 : Bool;
      b825 : Bool;
      b826 : Bool;
      b827 : Bool;
      b830 : Bool;
      b831 : Bool;
      b832 : Bool;
      b833 : Bool;
      b834 : Bool;
      b835 : Bool;
      b836 : Bool;
      b837 : Bool;
      b840 : Bool;
      b841 : Bool;
      b842 : Bool;
      b843 : Bool;
      b844 : Bool;
      b845 : Bool;
      b846 : Bool;
      b847 : Bool;
      b850 : Bool;
      b851 : Bool;
      b852 : Bool;
      b853 : Bool;
      b854 : Bool;
      b855 : Bool;
      b856 : Bool;
      b857 : Bool;
      b860 : Bool;
      b861 : Bool;
      b862 : Bool;
      b863 : Bool;
      b864 : Bool;
      b865 : Bool;
      b866 : Bool;
      b867 : Bool;
      b870 : Bool;
      b871 : Bool;
      b872 : Bool;
      b873 : Bool;
      b874 : Bool;
      b875 : Bool;
      b876 : Bool;
      b877 : Bool;
      b880 : Bool;
      b881 : Bool;
      b882 : Bool;
      b883 : Bool;
      b884 : Bool;
      b885 : Bool;
      b886 : Bool;
      b887 : Bool;
      b890 : Bool;
      b891 : Bool;
      b892 : Bool;
      b893 : Bool;
      b894 : Bool;
      b895 : Bool;
      b896 : Bool;
      b897 : Bool;
      b900 : Bool;
      b901 : Bool;
      b902 : Bool;
      b903 : Bool;
      b904 : Bool;
      b905 : Bool;
      b906 : Bool;
      b907 : Bool;
      b910 : Bool;
      b911 : Bool;
      b912 : Bool;
      b913 : Bool;
      b914 : Bool;
      b915 : Bool;
      b916 : Bool;
      b917 : Bool;
      b920 : Bool;
      b921 : Bool;
      b922 : Bool;
      b923 : Bool;
      b924 : Bool;
      b925 : Bool;
      b926 : Bool;
      b927 : Bool;
      b930 : Bool;
      b931 : Bool;
      b932 : Bool;
      b933 : Bool;
      b934 : Bool;
      b935 : Bool;
      b936 : Bool;
      b937 : Bool;
      b940 : Bool;
      b941 : Bool;
      b942 : Bool;
      b943 : Bool;
      b944 : Bool;
      b945 : Bool;
      b946 : Bool;
      b947 : Bool;
      b950 : Bool;
      b951 : Bool;
      b952 : Bool;
      b953 : Bool;
      b954 : Bool;
      b955 : Bool;
      b956 : Bool;
      b957 : Bool;
      b960 : Bool;
      b961 : Bool;
      b962 : Bool;
      b963 : Bool;
      b964 : Bool;
      b965 : Bool;
      b966 : Bool;
      b967 : Bool;
      b970 : Bool;
      b971 : Bool;
      b972 : Bool;
      b973 : Bool;
      b974 : Bool;
      b975 : Bool;
      b976 : Bool;
      b977 : Bool;
      b980 : Bool;
      b981 : Bool;
      b982 : Bool;
      b983 : Bool;
      b984 : Bool;
      b985 : Bool;
      b986 : Bool;
      b987 : Bool;
      b990 : Bool;
      b991 : Bool;
      b992 : Bool;
      b993 : Bool;
      b994 : Bool;
      b995 : Bool;
      b996 : Bool;
      b997 : Bool;
      b1000 : Bool;
      b1001 : Bool;
      b1002 : Bool;
      b1003 : Bool;
      b1004 : Bool;
      b1005 : Bool;
      b1006 : Bool;
      b1007 : Bool;
      b1010 : Bool;
      b1011 : Bool;
      b1012 : Bool;
      b1013 : Bool;
      b1014 : Bool;
      b1015 : Bool;
      b1016 : Bool;
      b1017 : Bool;
      b1020 : Bool;
      b1021 : Bool;
      b1022 : Bool;
      b1023 : Bool;
      b1024 : Bool;
      b1025 : Bool;
      b1026 : Bool;
      b1027 : Bool;
      b1030 : Bool;
      b1031 : Bool;
      b1032 : Bool;
      b1033 : Bool;
      b1034 : Bool;
      b1035 : Bool;
      b1036 : Bool;
      b1037 : Bool;
      b1040 : Bool;
      b1041 : Bool;
      b1042 : Bool;
      b1043 : Bool;
      b1044 : Bool;
      b1045 : Bool;
      b1046 : Bool;
      b1047 : Bool;
      b1050 : Bool;
      b1051 : Bool;
      b1052 : Bool;
      b1053 : Bool;
      b1054 : Bool;
      b1055 : Bool;
      b1056 : Bool;
      b1057 : Bool;
      b1060 : Bool;
      b1061 : Bool;
      b1062 : Bool;
      b1063 : Bool;
      b1064 : Bool;
      b1065 : Bool;
      b1066 : Bool;
      b1067 : Bool;
      b1070 : Bool;
      b1071 : Bool;
      b1072 : Bool;
      b1073 : Bool;
      b1074 : Bool;
      b1075 : Bool;
      b1076 : Bool;
      b1077 : Bool;
      b1080 : Bool;
      b1081 : Bool;
      b1082 : Bool;
      b1083 : Bool;
      b1084 : Bool;
      b1085 : Bool;
      b1086 : Bool;
      b1087 : Bool;
      b1090 : Bool;
      b1091 : Bool;
      b1092 : Bool;
      b1093 : Bool;
      b1094 : Bool;
      b1095 : Bool;
      b1096 : Bool;
      b1097 : Bool;
      b1100 : Bool;
      b1101 : Bool;
      b1102 : Bool;
      b1103 : Bool;
      b1104 : Bool;
      b1105 : Bool;
      b1106 : Bool;
      b1107 : Bool;
      b1110 : Bool;
      b1111 : Bool;
      b1112 : Bool;
      b1113 : Bool;
      b1114 : Bool;
      b1115 : Bool;
      b1116 : Bool;
      b1117 : Bool;
      b1120 : Bool;
      b1121 : Bool;
      b1122 : Bool;
      b1123 : Bool;
      b1124 : Bool;
      b1125 : Bool;
      b1126 : Bool;
      b1127 : Bool;
      b1130 : Bool;
      b1131 : Bool;
      b1132 : Bool;
      b1133 : Bool;
      b1134 : Bool;
      b1135 : Bool;
      b1136 : Bool;
      b1137 : Bool;
      b1140 : Bool;
      b1141 : Bool;
      b1142 : Bool;
      b1143 : Bool;
      b1144 : Bool;
      b1145 : Bool;
      b1146 : Bool;
      b1147 : Bool;
      b1150 : Bool;
      b1151 : Bool;
      b1152 : Bool;
      b1153 : Bool;
      b1154 : Bool;
      b1155 : Bool;
      b1156 : Bool;
      b1157 : Bool;
      b1160 : Bool;
      b1161 : Bool;
      b1162 : Bool;
      b1163 : Bool;
      b1164 : Bool;
      b1165 : Bool;
      b1166 : Bool;
      b1167 : Bool;
      b1170 : Bool;
      b1171 : Bool;
      b1172 : Bool;
      b1173 : Bool;
      b1174 : Bool;
      b1175 : Bool;
      b1176 : Bool;
      b1177 : Bool;
      b1180 : Bool;
      b1181 : Bool;
      b1182 : Bool;
      b1183 : Bool;
      b1184 : Bool;
      b1185 : Bool;
      b1186 : Bool;
      b1187 : Bool;
      b1190 : Bool;
      b1191 : Bool;
      b1192 : Bool;
      b1193 : Bool;
      b1194 : Bool;
      b1195 : Bool;
      b1196 : Bool;
      b1197 : Bool;
      b1200 : Bool;
      b1201 : Bool;
      b1202 : Bool;
      b1203 : Bool;
      b1204 : Bool;
      b1205 : Bool;
      b1206 : Bool;
      b1207 : Bool;
      b1210 : Bool;
      b1211 : Bool;
      b1212 : Bool;
      b1213 : Bool;
      b1214 : Bool;
      b1215 : Bool;
      b1216 : Bool;
      b1217 : Bool;
      b1220 : Bool;
      b1221 : Bool;
      b1222 : Bool;
      b1223 : Bool;
      b1224 : Bool;
      b1225 : Bool;
      b1226 : Bool;
      b1227 : Bool;
      b1230 : Bool;
      b1231 : Bool;
      b1232 : Bool;
      b1233 : Bool;
      b1234 : Bool;
      b1235 : Bool;
      b1236 : Bool;
      b1237 : Bool;
      b1240 : Bool;
      b1241 : Bool;
      b1242 : Bool;
      b1243 : Bool;
      b1244 : Bool;
      b1245 : Bool;
      b1246 : Bool;
      b1247 : Bool;
      b1250 : Bool;
      b1251 : Bool;
      b1252 : Bool;
      b1253 : Bool;
      b1254 : Bool;
      b1255 : Bool;
      b1256 : Bool;
      b1257 : Bool;
      b1260 : Bool;
      b1261 : Bool;
      b1262 : Bool;
      b1263 : Bool;
      b1264 : Bool;
      b1265 : Bool;
      b1266 : Bool;
      b1267 : Bool;
      b1270 : Bool;
      b1271 : Bool;
      b1272 : Bool;
      b1273 : Bool;
      b1274 : Bool;
      b1275 : Bool;
      b1276 : Bool;
      b1277 : Bool;
      b1280 : Bool;
      b1281 : Bool;
      b1282 : Bool;
      b1283 : Bool;
      b1284 : Bool;
      b1285 : Bool;
      b1286 : Bool;
      b1287 : Bool;
      b1290 : Bool;
      b1291 : Bool;
      b1292 : Bool;
      b1293 : Bool;
      b1294 : Bool;
      b1295 : Bool;
      b1296 : Bool;
      b1297 : Bool;
      b1300 : Bool;
      b1301 : Bool;
      b1302 : Bool;
      b1303 : Bool;
      b1304 : Bool;
      b1305 : Bool;
      b1306 : Bool;
      b1307 : Bool;
      b1310 : Bool;
      b1311 : Bool;
      b1312 : Bool;
      b1313 : Bool;
      b1314 : Bool;
      b1315 : Bool;
      b1316 : Bool;
      b1317 : Bool;
      b1320 : Bool;
      b1321 : Bool;
      b1322 : Bool;
      b1323 : Bool;
      b1324 : Bool;
      b1325 : Bool;
      b1326 : Bool;
      b1327 : Bool;
      b1330 : Bool;
      b1331 : Bool;
      b1332 : Bool;
      b1333 : Bool;
      b1334 : Bool;
      b1335 : Bool;
      b1336 : Bool;
      b1337 : Bool;
      b1340 : Bool;
      b1341 : Bool;
      b1342 : Bool;
      b1343 : Bool;
      b1344 : Bool;
      b1345 : Bool;
      b1346 : Bool;
      b1347 : Bool;
      b1350 : Bool;
      b1351 : Bool;
      b1352 : Bool;
      b1353 : Bool;
      b1354 : Bool;
      b1355 : Bool;
      b1356 : Bool;
      b1357 : Bool;
      b1360 : Bool;
      b1361 : Bool;
      b1362 : Bool;
      b1363 : Bool;
      b1364 : Bool;
      b1365 : Bool;
      b1366 : Bool;
      b1367 : Bool;
      b1370 : Bool;
      b1371 : Bool;
      b1372 : Bool;
      b1373 : Bool;
      b1374 : Bool;
      b1375 : Bool;
      b1376 : Bool;
      b1377 : Bool;
      b1380 : Bool;
      b1381 : Bool;
      b1382 : Bool;
      b1383 : Bool;
      b1384 : Bool;
      b1385 : Bool;
      b1386 : Bool;
      b1387 : Bool;
      b1390 : Bool;
      b1391 : Bool;
      b1392 : Bool;
      b1393 : Bool;
      b1394 : Bool;
      b1395 : Bool;
      b1396 : Bool;
      b1397 : Bool;
      b1400 : Bool;
      b1401 : Bool;
      b1402 : Bool;
      b1403 : Bool;
      b1404 : Bool;
      b1405 : Bool;
      b1406 : Bool;
      b1407 : Bool;
      b1410 : Bool;
      b1411 : Bool;
      b1412 : Bool;
      b1413 : Bool;
      b1414 : Bool;
      b1415 : Bool;
      b1416 : Bool;
      b1417 : Bool;
      b1420 : Bool;
      b1421 : Bool;
      b1422 : Bool;
      b1423 : Bool;
      b1424 : Bool;
      b1425 : Bool;
      b1426 : Bool;
      b1427 : Bool;
      b1430 : Bool;
      b1431 : Bool;
      b1432 : Bool;
      b1433 : Bool;
      b1434 : Bool;
      b1435 : Bool;
      b1436 : Bool;
      b1437 : Bool;
      b1440 : Bool;
      b1441 : Bool;
      b1442 : Bool;
      b1443 : Bool;
      b1444 : Bool;
      b1445 : Bool;
      b1446 : Bool;
      b1447 : Bool;
      b1450 : Bool;
      b1451 : Bool;
      b1452 : Bool;
      b1453 : Bool;
      b1454 : Bool;
      b1455 : Bool;
      b1456 : Bool;
      b1457 : Bool;
      b1460 : Bool;
      b1461 : Bool;
      b1462 : Bool;
      b1463 : Bool;
      b1464 : Bool;
      b1465 : Bool;
      b1466 : Bool;
      b1467 : Bool;
      b1470 : Bool;
      b1471 : Bool;
      b1472 : Bool;
      b1473 : Bool;
      b1474 : Bool;
      b1475 : Bool;
      b1476 : Bool;
      b1477 : Bool;
      b1480 : Bool;
      b1481 : Bool;
      b1482 : Bool;
      b1483 : Bool;
      b1484 : Bool;
      b1485 : Bool;
      b1486 : Bool;
      b1487 : Bool;
      b1490 : Bool;
      b1491 : Bool;
      b1492 : Bool;
      b1493 : Bool;
      b1494 : Bool;
      b1495 : Bool;
      b1496 : Bool;
      b1497 : Bool;
      M338 : Bool;
      b1501 : Bool;
      b1502 : Bool;
      b1503 : Bool;
      b1504 : Bool;
      b1505 : Bool;
      b1506 : Bool;
      b1507 : Bool;
      b1510 : Bool;
      b1511 : Bool;
      b1512 : Bool;
      b1513 : Bool;
      b1514 : Bool;
      b1515 : Bool;
      b1516 : Bool;
      b1517 : Bool;
      b1520 : Bool;
      b1521 : Bool;
      b1522 : Bool;
      b1523 : Bool;
      b1524 : Bool;
      b1525 : Bool;
      b1526 : Bool;
      b1527 : Bool;
      b1530 : Bool;
      b1531 : Bool;
      b1532 : Bool;
      b1533 : Bool;
      b1534 : Bool;
      b1535 : Bool;
      b1536 : Bool;
      b1537 : Bool;
      b1540 : Bool;
      b1541 : Bool;
      b1542 : Bool;
      b1543 : Bool;
      b1544 : Bool;
      b1545 : Bool;
      b1546 : Bool;
      b1547 : Bool;
      b1550 : Bool;
      b1551 : Bool;
      b1552 : Bool;
      b1553 : Bool;
      b1554 : Bool;
      b1555 : Bool;
      b1556 : Bool;
      b1557 : Bool;
      b1560 : Bool;
      b1561 : Bool;
      b1562 : Bool;
      b1563 : Bool;
      b1564 : Bool;
      b1565 : Bool;
      b1566 : Bool;
      b1567 : Bool;
      b1570 : Bool;
      b1571 : Bool;
      b1572 : Bool;
      b1573 : Bool;
      b1574 : Bool;
      b1575 : Bool;
      b1576 : Bool;
      b1577 : Bool;
      b1580 : Bool;
      b1581 : Bool;
      b1582 : Bool;
      b1583 : Bool;
      b1584 : Bool;
      b1585 : Bool;
      b1586 : Bool;
      b1587 : Bool;
      b1590 : Bool;
      b1591 : Bool;
      b1592 : Bool;
      b1593 : Bool;
      b1594 : Bool;
      b1595 : Bool;
      b1596 : Bool;
      b1597 : Bool;
      b1600 : Bool;
      b1601 : Bool;
      b1602 : Bool;
      b1603 : Bool;
      b1604 : Bool;
      b1605 : Bool;
      b1606 : Bool;
      b1607 : Bool;
      b1610 : Bool;
      b1611 : Bool;
      b1612 : Bool;
      b1613 : Bool;
      b1614 : Bool;
      b1615 : Bool;
      b1616 : Bool;
      b1617 : Bool;
      b1620 : Bool;
      b1621 : Bool;
      b1622 : Bool;
      b1623 : Bool;
      b1624 : Bool;
      b1625 : Bool;
      b1626 : Bool;
      b1627 : Bool;
      b1630 : Bool;
      b1631 : Bool;
      b1632 : Bool;
      b1633 : Bool;
      b1634 : Bool;
      b1635 : Bool;
      b1636 : Bool;
      b1637 : Bool;
      b1640 : Bool;
      b1641 : Bool;
      b1642 : Bool;
      b1643 : Bool;
      b1644 : Bool;
      b1645 : Bool;
      b1646 : Bool;
      b1647 : Bool;
      b1650 : Bool;
      b1651 : Bool;
      b1652 : Bool;
      b1653 : Bool;
      b1654 : Bool;
      b1655 : Bool;
      b1656 : Bool;
      b1657 : Bool;
      b1660 : Bool;
      b1661 : Bool;
      b1662 : Bool;
      b1663 : Bool;
      b1664 : Bool;
      b1665 : Bool;
      b1666 : Bool;
      b1667 : Bool;
      b1670 : Bool;
      b1671 : Bool;
      b1672 : Bool;
      b1673 : Bool;
      b1674 : Bool;
      b1675 : Bool;
      b1676 : Bool;
      b1677 : Bool;
      b1680 : Bool;
      b1681 : Bool;
      b1682 : Bool;
      b1683 : Bool;
      b1684 : Bool;
      b1685 : Bool;
      b1686 : Bool;
      b1687 : Bool;
      b1690 : Bool;
      b1691 : Bool;
      b1692 : Bool;
      b1693 : Bool;
      b1694 : Bool;
      b1695 : Bool;
      b1696 : Bool;
      b1697 : Bool;
      b1700 : Bool;
      b1701 : Bool;
      b1702 : Bool;
      b1703 : Bool;
      b1704 : Bool;
      b1705 : Bool;
      b1706 : Bool;
      b1707 : Bool;
      b1710 : Bool;
      b1711 : Bool;
      b1712 : Bool;
      b1713 : Bool;
      b1714 : Bool;
      b1715 : Bool;
      b1716 : Bool;
      b1717 : Bool;
      b1720 : Bool;
      b1721 : Bool;
      b1722 : Bool;
      b1723 : Bool;
      b1724 : Bool;
      b1725 : Bool;
      b1726 : Bool;
      b1727 : Bool;
      b1730 : Bool;
      b1731 : Bool;
      b1732 : Bool;
      b1733 : Bool;
      b1734 : Bool;
      b1735 : Bool;
      b1736 : Bool;
      b1737 : Bool;
      b1740 : Bool;
      b1741 : Bool;
      b1742 : Bool;
      b1743 : Bool;
      b1744 : Bool;
      b1745 : Bool;
      b1746 : Bool;
      b1747 : Bool;
      b1750 : Bool;
      b1751 : Bool;
      b1752 : Bool;
      b1753 : Bool;
      b1754 : Bool;
      b1755 : Bool;
      b1756 : Bool;
      b1757 : Bool;
      b1760 : Bool;
      b1761 : Bool;
      b1762 : Bool;
      b1763 : Bool;
      b1764 : Bool;
      b1765 : Bool;
      b1766 : Bool;
      b1767 : Bool;
      b1770 : Bool;
      b1771 : Bool;
      b1772 : Bool;
      b1773 : Bool;
      b1774 : Bool;
      b1775 : Bool;
      b1776 : Bool;
      b1777 : Bool;
      b1780 : Bool;
      b1781 : Bool;
      b1782 : Bool;
      b1783 : Bool;
      b1784 : Bool;
      b1785 : Bool;
      b1786 : Bool;
      b1787 : Bool;
      b1790 : Bool;
      b1791 : Bool;
      b1792 : Bool;
      b1793 : Bool;
      b1794 : Bool;
      b1795 : Bool;
      b1796 : Bool;
      b1797 : Bool;
      b1800 : Bool;
      b1801 : Bool;
      b1802 : Bool;
      b1803 : Bool;
      b1804 : Bool;
      b1805 : Bool;
      b1806 : Bool;
      b1807 : Bool;
      b1810 : Bool;
      b1811 : Bool;
      b1812 : Bool;
      b1813 : Bool;
      b1814 : Bool;
      b1815 : Bool;
      b1816 : Bool;
      b1817 : Bool;
      b1820 : Bool;
      b1821 : Bool;
      b1822 : Bool;
      b1823 : Bool;
      b1824 : Bool;
      b1825 : Bool;
      b1826 : Bool;
      b1827 : Bool;
      b1830 : Bool;
      b1831 : Bool;
      b1832 : Bool;
      b1833 : Bool;
      b1834 : Bool;
      b1835 : Bool;
      b1836 : Bool;
      b1837 : Bool;
      b1840 : Bool;
      b1841 : Bool;
      b1842 : Bool;
      b1843 : Bool;
      b1844 : Bool;
      b1845 : Bool;
      b1846 : Bool;
      b1847 : Bool;
      b1850 : Bool;
      b1851 : Bool;
      b1852 : Bool;
      b1853 : Bool;
      b1854 : Bool;
      b1855 : Bool;
      b1856 : Bool;
      b1857 : Bool;
      b1860 : Bool;
      b1861 : Bool;
      b1862 : Bool;
      b1863 : Bool;
      b1864 : Bool;
      b1865 : Bool;
      b1866 : Bool;
      b1867 : Bool;
      b1870 : Bool;
      b1871 : Bool;
      b1872 : Bool;
      b1873 : Bool;
      b1874 : Bool;
      b1875 : Bool;
      b1876 : Bool;
      b1877 : Bool;
      b1880 : Bool;
      b1881 : Bool;
      b1882 : Bool;
      b1883 : Bool;
      b1884 : Bool;
      b1885 : Bool;
      b1886 : Bool;
      b1887 : Bool;
      b1890 : Bool;
      b1891 : Bool;
      b1892 : Bool;
      b1893 : Bool;
      b1894 : Bool;
      b1895 : Bool;
      b1896 : Bool;
      b1897 : Bool;
   END_STRUCT;


BEGIN
   b40 := TRUE;
   b182 := TRUE;
   b184 := TRUE;
   b192 := TRUE;
   b194 := TRUE;
   b320 := TRUE;
   b322 := TRUE;
   b326 := TRUE;
   b720 := TRUE;
   b721 := TRUE;
   b727 := TRUE;
   b770 := TRUE;
   b772 := TRUE;
   b782 := TRUE;
   b783 := TRUE;
   b784 := TRUE;
   b785 := TRUE;
   b801 := TRUE;
   b1301 := TRUE;
   b1321 := TRUE;
   b1323 := TRUE;
   b1325 := TRUE;
   b1326 := TRUE;
   b1404 := TRUE;
   b1464 := TRUE;
   b1480 := TRUE;
   b1542 := TRUE;
   b1550 := TRUE;
   b1582 := TRUE;
   b1590 := TRUE;

END_DATA_BLOCK

